Universal Robots URScript: test-1.urscript

def tuft_program():
    global tuft_coords = p[-0.743799, 1.270828, -0.183331, 1.574839, 0.004352, -0.002073]
    global current_pose = p[0,0,0,-1.19353,1.19941,1.24224]
    textmsg("Starting tufting job test-1.jpg")
    textmsg("Using coordinate frame tuft_coords")
    set_digital_out(0, False)
    global travel_speed = 0.2000
    global tuft_speed = 0.0600
    global contact_force_threshold = 15.00
    global contact_probe_step = 0.0010
    global progress_host = "127.0.0.1"
    global progress_port = 4700
    global progress_total = 2256
    global progress_current = 0
    global progress_job_id = "645c90bf-1acd-4e3e-9f73-d32fedb47cbd"
    global open=socket_open(progress_host,progress_port)
    while (open ==  False  ):
        global open=socket_open(progress_host,progress_port)
    end
    def report_progress():
        progress_current = progress_current + 1
        global sendToServer="{jobId:" + progress_job_id + ",current:" + to_str(progress_current) + ",total:" + to_str(progress_total) + "}
"
        socket_send_string(sendToServer)
    end
    new_pose = pose_trans(tuft_coords, p[0.3854, 0.5062, 0.1500, 0, 0, 0])
    movel(p[new_pose[0], new_pose[1], new_pose[2], current_pose[3], current_pose[4], current_pose[5]], a=1.2, v=0.2000)
    report_progress()
    new_pose = pose_trans(tuft_coords, p[0.3854, 0.5062, -0.0020, 0, 0, 0])
    movel(p[new_pose[0], new_pose[1], new_pose[2], current_pose[3], current_pose[4], current_pose[5]], a=0.8, v=0.2000)
    report_progress()
    set_digital_out(0, True)
    new_pose = pose_trans(tuft_coords, p[0.3854, 0.5438, -0.0020, 0, 0, 0])
    movel(p[new_pose[0], new_pose[1], new_pose[2], current_pose[3], current_pose[4], current_pose[5]], a=1.2, v=0.0600)
    report_progress()
    set_digital_out(0, False)
    new_pose = pose_trans(tuft_coords, p[0.3854, 0.5438, 0.1500, 0, 0, 0])
    movel(p[new_pose[0], new_pose[1], new_pose[2], current_pose[3], current_pose[4], current_pose[5]], a=0.8, v=0.2000)
    report_progress()
    new_pose = pose_trans(tuft_coords, p[0.3874, 0.4824, 0.1500, 0, 0, 0])
    movel(p[new_pose[0], new_pose[1], new_pose[2], current_pose[3], current_pose[4], current_pose[5]], a=1.2, v=0.2000)
    report_progress()
    new_pose = pose_trans(tuft_coords, p[0.3874, 0.4824, -0.0020, 0, 0, 0])
    movel(p[new_pose[0], new_pose[1], new_pose[2], current_pose[3], current_pose[4], current_pose[5]], a=0.8, v=0.2000)
    report_progress()
    set_digital_out(0, True)
    new_pose = pose_trans(tuft_coords, p[0.3874, 0.5676, -0.0020, 0, 0, 0])
    movel(p[new_pose[0], new_pose[1], new_pose[2], current_pose[3], current_pose[4], current_pose[5]], a=1.2, v=0.0600)
    report_progress()
    set_digital_out(0, False)
    new_pose = pose_trans(tuft_coords, p[0.3874, 0.5676, 0.1500, 0, 0, 0])
    movel(p[new_pose[0], new_pose[1], new_pose[2], current_pose[3], current_pose[4], current_pose[5]], a=0.8, v=0.2000)
    report_progress()
    new_pose = pose_trans(tuft_coords, p[0.3893, 0.4686, 0.1500, 0, 0, 0])
    movel(p[new_pose[0], new_pose[1], new_pose[2], current_pose[3], current_pose[4], current_pose[5]], a=1.2, v=0.2000)
    report_progress()
    new_pose = pose_trans(tuft_coords, p[0.3893, 0.4686, -0.0020, 0, 0, 0])
    movel(p[new_pose[0], new_pose[1], new_pose[2], current_pose[3], current_pose[4], current_pose[5]], a=0.8, v=0.2000)
    report_progress()
    set_digital_out(0, True)
    new_pose = pose_trans(tuft_coords, p[0.3893, 0.5814, -0.0020, 0, 0, 0])
    movel(p[new_pose[0], new_pose[1], new_pose[2], current_pose[3], current_pose[4], current_pose[5]], a=1.2, v=0.0600)
    report_progress()
    set_digital_out(0, False)
    new_pose = pose_trans(tuft_coords, p[0.3893, 0.5814, 0.1500, 0, 0, 0])
    movel(p[new_pose[0], new_pose[1], new_pose[2], current_pose[3], current_pose[4], current_pose[5]], a=0.8, v=0.2000)
    report_progress()
    new_pose = pose_trans(tuft_coords, p[0.3912, 0.4567, 0.1500, 0, 0, 0])
    movel(p[new_pose[0], new_pose[1], new_pose[2], current_pose[3], current_pose[4], current_pose[5]], a=1.2, v=0.2000)
    report_progress()
    new_pose = pose_trans(tuft_coords, p[0.3912, 0.4567, -0.0020, 0, 0, 0])
    movel(p[new_pose[0], new_pose[1], new_pose[2], current_pose[3], current_pose[4], current_pose[5]], a=0.8, v=0.2000)
    report_progress()
    set_digital_out(0, True)
    new_pose = pose_trans(tuft_coords, p[0.3912, 0.5933, -0.0020, 0, 0, 0])
    movel(p[new_pose[0], new_pose[1], new_pose[2], current_pose[3], current_pose[4], current_pose[5]], a=1.2, v=0.0600)
    report_progress()
    set_digital_out(0, False)
    new_pose = pose_trans(tuft_coords, p[0.3912, 0.5933, 0.1500, 0, 0, 0])
    movel(p[new_pose[0], new_pose[1], new_pose[2], current_pose[3], current_pose[4], current_pose[5]], a=0.8, v=0.2000)
    report_progress()
    new_pose = pose_trans(tuft_coords, p[0.3932, 0.4468, 0.1500, 0, 0, 0])
    movel(p[new_pose[0], new_pose[1], new_pose[2], current_pose[3], current_pose[4], current_pose[5]], a=1.2, v=0.2000)
    report_progress()
    new_pose = pose_trans(tuft_coords, p[0.3932, 0.4468, -0.0020, 0, 0, 0])
    movel(p[new_pose[0], new_pose[1], new_pose[2], current_pose[3], current_pose[4], current_pose[5]], a=0.8, v=0.2000)
    report_progress()
    set_digital_out(0, True)
    new_pose = pose_trans(tuft_coords, p[0.3932, 0.6032, -0.0020, 0, 0, 0])
    movel(p[new_pose[0], new_pose[1], new_pose[2], current_pose[3], current_pose[4], current_pose[5]], a=1.2, v=0.0600)
    report_progress()
    set_digital_out(0, False)
    new_pose = pose_trans(tuft_coords, p[0.3932, 0.6032, 0.1500, 0, 0, 0])
    movel(p[new_pose[0], new_pose[1], new_pose[2], current_pose[3], current_pose[4], current_pose[5]], a=0.8, v=0.2000)
    report_progress()
    new_pose = pose_trans(tuft_coords, p[0.3951, 0.4389, 0.1500, 0, 0, 0])
    movel(p[new_pose[0], new_pose[1], new_pose[2], current_pose[3], current_pose[4], current_pose[5]], a=1.2, v=0.2000)
    report_progress()
    new_pose = pose_trans(tuft_coords, p[0.3951, 0.4389, -0.0020, 0, 0, 0])
    movel(p[new_pose[0], new_pose[1], new_pose[2], current_pose[3], current_pose[4], current_pose[5]], a=0.8, v=0.2000)
    report_progress()
    set_digital_out(0, True)
    new_pose = pose_trans(tuft_coords, p[0.3951, 0.6111, -0.0020, 0, 0, 0])
    movel(p[new_pose[0], new_pose[1], new_pose[2], current_pose[3], current_pose[4], current_pose[5]], a=1.2, v=0.0600)
    report_progress()
    set_digital_out(0, False)
    new_pose = pose_trans(tuft_coords, p[0.3951, 0.6111, 0.1500, 0, 0, 0])
    movel(p[new_pose[0], new_pose[1], new_pose[2], current_pose[3], current_pose[4], current_pose[5]], a=0.8, v=0.2000)
    report_progress()
    new_pose = pose_trans(tuft_coords, p[0.3971, 0.4310, 0.1500, 0, 0, 0])
    movel(p[new_pose[0], new_pose[1], new_pose[2], current_pose[3], current_pose[4], current_pose[5]], a=1.2, v=0.2000)
    report_progress()
    new_pose = pose_trans(tuft_coords, p[0.3971, 0.4310, -0.0020, 0, 0, 0])
    movel(p[new_pose[0], new_pose[1], new_pose[2], current_pose[3], current_pose[4], current_pose[5]], a=0.8, v=0.2000)
    report_progress()
    set_digital_out(0, True)
    new_pose = pose_trans(tuft_coords, p[0.3971, 0.6190, -0.0020, 0, 0, 0])
    movel(p[new_pose[0], new_pose[1], new_pose[2], current_pose[3], current_pose[4], current_pose[5]], a=1.2, v=0.0600)
    report_progress()
    set_digital_out(0, False)
    new_pose = pose_trans(tuft_coords, p[0.3971, 0.6190, 0.1500, 0, 0, 0])
    movel(p[new_pose[0], new_pose[1], new_pose[2], current_pose[3], current_pose[4], current_pose[5]], a=0.8, v=0.2000)
    report_progress()
    new_pose = pose_trans(tuft_coords, p[0.3990, 0.4231, 0.1500, 0, 0, 0])
    movel(p[new_pose[0], new_pose[1], new_pose[2], current_pose[3], current_pose[4], current_pose[5]], a=1.2, v=0.2000)
    report_progress()
    new_pose = pose_trans(tuft_coords, p[0.3990, 0.4231, -0.0020, 0, 0, 0])
    movel(p[new_pose[0], new_pose[1], new_pose[2], current_pose[3], current_pose[4], current_pose[5]], a=0.8, v=0.2000)
    report_progress()
    set_digital_out(0, True)
    new_pose = pose_trans(tuft_coords, p[0.3990, 0.6269, -0.0020, 0, 0, 0])
    movel(p[new_pose[0], new_pose[1], new_pose[2], current_pose[3], current_pose[4], current_pose[5]], a=1.2, v=0.0600)
    report_progress()
    set_digital_out(0, False)
    new_pose = pose_trans(tuft_coords, p[0.3990, 0.6269, 0.1500, 0, 0, 0])
    movel(p[new_pose[0], new_pose[1], new_pose[2], current_pose[3], current_pose[4], current_pose[5]], a=0.8, v=0.2000)
    report_progress()
    new_pose = pose_trans(tuft_coords, p[0.4010, 0.4171, 0.1500, 0, 0, 0])
    movel(p[new_pose[0], new_pose[1], new_pose[2], current_pose[3], current_pose[4], current_pose[5]], a=1.2, v=0.2000)
    report_progress()
    new_pose = pose_trans(tuft_coords, p[0.4010, 0.4171, -0.0020, 0, 0, 0])
    movel(p[new_pose[0], new_pose[1], new_pose[2], current_pose[3], current_pose[4], current_pose[5]], a=0.8, v=0.2000)
    report_progress()
    set_digital_out(0, True)
    new_pose = pose_trans(tuft_coords, p[0.4010, 0.6329, -0.0020, 0, 0, 0])
    movel(p[new_pose[0], new_pose[1], new_pose[2], current_pose[3], current_pose[4], current_pose[5]], a=1.2, v=0.0600)
    report_progress()
    set_digital_out(0, False)
    new_pose = pose_trans(tuft_coords, p[0.4010, 0.6329, 0.1500, 0, 0, 0])
    movel(p[new_pose[0], new_pose[1], new_pose[2], current_pose[3], current_pose[4], current_pose[5]], a=0.8, v=0.2000)
    report_progress()
    new_pose = pose_trans(tuft_coords, p[0.4029, 0.4112, 0.1500, 0, 0, 0])
    movel(p[new_pose[0], new_pose[1], new_pose[2], current_pose[3], current_pose[4], current_pose[5]], a=1.2, v=0.2000)
    report_progress()
    new_pose = pose_trans(tuft_coords, p[0.4029, 0.4112, -0.0020, 0, 0, 0])
    movel(p[new_pose[0], new_pose[1], new_pose[2], current_pose[3], current_pose[4], current_pose[5]], a=0.8, v=0.2000)
    report_progress()
    set_digital_out(0, True)
    new_pose = pose_trans(tuft_coords, p[0.4029, 0.6388, -0.0020, 0, 0, 0])
    movel(p[new_pose[0], new_pose[1], new_pose[2], current_pose[3], current_pose[4], current_pose[5]], a=1.2, v=0.0600)
    report_progress()
    set_digital_out(0, False)
    new_pose = pose_trans(tuft_coords, p[0.4029, 0.6388, 0.1500, 0, 0, 0])
    movel(p[new_pose[0], new_pose[1], new_pose[2], current_pose[3], current_pose[4], current_pose[5]], a=0.8, v=0.2000)
    report_progress()
    new_pose = pose_trans(tuft_coords, p[0.4049, 0.4053, 0.1500, 0, 0, 0])
    movel(p[new_pose[0], new_pose[1], new_pose[2], current_pose[3], current_pose[4], current_pose[5]], a=1.2, v=0.2000)
    report_progress()
    new_pose = pose_trans(tuft_coords, p[0.4049, 0.4053, -0.0020, 0, 0, 0])
    movel(p[new_pose[0], new_pose[1], new_pose[2], current_pose[3], current_pose[4], current_pose[5]], a=0.8, v=0.2000)
    report_progress()
    set_digital_out(0, True)
    new_pose = pose_trans(tuft_coords, p[0.4049, 0.6447, -0.0020, 0, 0, 0])
    movel(p[new_pose[0], new_pose[1], new_pose[2], current_pose[3], current_pose[4], current_pose[5]], a=1.2, v=0.0600)
    report_progress()
    set_digital_out(0, False)
    new_pose = pose_trans(tuft_coords, p[0.4049, 0.6447, 0.1500, 0, 0, 0])
    movel(p[new_pose[0], new_pose[1], new_pose[2], current_pose[3], current_pose[4], current_pose[5]], a=0.8, v=0.2000)
    report_progress()
    new_pose = pose_trans(tuft_coords, p[0.4068, 0.3993, 0.1500, 0, 0, 0])
    movel(p[new_pose[0], new_pose[1], new_pose[2], current_pose[3], current_pose[4], current_pose[5]], a=1.2, v=0.2000)
    report_progress()
    new_pose = pose_trans(tuft_coords, p[0.4068, 0.3993, -0.0020, 0, 0, 0])
    movel(p[new_pose[0], new_pose[1], new_pose[2], current_pose[3], current_pose[4], current_pose[5]], a=0.8, v=0.2000)
    report_progress()
    set_digital_out(0, True)
    new_pose = pose_trans(tuft_coords, p[0.4068, 0.6507, -0.0020, 0, 0, 0])
    movel(p[new_pose[0], new_pose[1], new_pose[2], current_pose[3], current_pose[4], current_pose[5]], a=1.2, v=0.0600)
    report_progress()
    set_digital_out(0, False)
    new_pose = pose_trans(tuft_coords, p[0.4068, 0.6507, 0.1500, 0, 0, 0])
    movel(p[new_pose[0], new_pose[1], new_pose[2], current_pose[3], current_pose[4], current_pose[5]], a=0.8, v=0.2000)
    report_progress()
    new_pose = pose_trans(tuft_coords, p[0.4088, 0.3934, 0.1500, 0, 0, 0])
    movel(p[new_pose[0], new_pose[1], new_pose[2], current_pose[3], current_pose[4], current_pose[5]], a=1.2, v=0.2000)
    report_progress()
    new_pose = pose_trans(tuft_coords, p[0.4088, 0.3934, -0.0020, 0, 0, 0])
    movel(p[new_pose[0], new_pose[1], new_pose[2], current_pose[3], current_pose[4], current_pose[5]], a=0.8, v=0.2000)
    report_progress()
    set_digital_out(0, True)
    new_pose = pose_trans(tuft_coords, p[0.4088, 0.6566, -0.0020, 0, 0, 0])
    movel(p[new_pose[0], new_pose[1], new_pose[2], current_pose[3], current_pose[4], current_pose[5]], a=1.2, v=0.0600)
    report_progress()
    set_digital_out(0, False)
    new_pose = pose_trans(tuft_coords, p[0.4088, 0.6566, 0.1500, 0, 0, 0])
    movel(p[new_pose[0], new_pose[1], new_pose[2], current_pose[3], current_pose[4], current_pose[5]], a=0.8, v=0.2000)
    report_progress()
    new_pose = pose_trans(tuft_coords, p[0.4107, 0.3874, 0.1500, 0, 0, 0])
    movel(p[new_pose[0], new_pose[1], new_pose[2], current_pose[3], current_pose[4], current_pose[5]], a=1.2, v=0.2000)
    report_progress()
    new_pose = pose_trans(tuft_coords, p[0.4107, 0.3874, -0.0020, 0, 0, 0])
    movel(p[new_pose[0], new_pose[1], new_pose[2], current_pose[3], current_pose[4], current_pose[5]], a=0.8, v=0.2000)
    report_progress()
    set_digital_out(0, True)
    new_pose = pose_trans(tuft_coords, p[0.4107, 0.6606, -0.0020, 0, 0, 0])
    movel(p[new_pose[0], new_pose[1], new_pose[2], current_pose[3], current_pose[4], current_pose[5]], a=1.2, v=0.0600)
    report_progress()
    set_digital_out(0, False)
    new_pose = pose_trans(tuft_coords, p[0.4107, 0.6606, 0.1500, 0, 0, 0])
    movel(p[new_pose[0], new_pose[1], new_pose[2], current_pose[3], current_pose[4], current_pose[5]], a=0.8, v=0.2000)
    report_progress()
    new_pose = pose_trans(tuft_coords, p[0.4126, 0.3835, 0.1500, 0, 0, 0])
    movel(p[new_pose[0], new_pose[1], new_pose[2], current_pose[3], current_pose[4], current_pose[5]], a=1.2, v=0.2000)
    report_progress()
    new_pose = pose_trans(tuft_coords, p[0.4126, 0.3835, -0.0020, 0, 0, 0])
    movel(p[new_pose[0], new_pose[1], new_pose[2], current_pose[3], current_pose[4], current_pose[5]], a=0.8, v=0.2000)
    report_progress()
    set_digital_out(0, True)
    new_pose = pose_trans(tuft_coords, p[0.4126, 0.6665, -0.0020, 0, 0, 0])
    movel(p[new_pose[0], new_pose[1], new_pose[2], current_pose[3], current_pose[4], current_pose[5]], a=1.2, v=0.0600)
    report_progress()
    set_digital_out(0, False)
    new_pose = pose_trans(tuft_coords, p[0.4126, 0.6665, 0.1500, 0, 0, 0])
    movel(p[new_pose[0], new_pose[1], new_pose[2], current_pose[3], current_pose[4], current_pose[5]], a=0.8, v=0.2000)
    report_progress()
    new_pose = pose_trans(tuft_coords, p[0.4146, 0.3795, 0.1500, 0, 0, 0])
    movel(p[new_pose[0], new_pose[1], new_pose[2], current_pose[3], current_pose[4], current_pose[5]], a=1.2, v=0.2000)
    report_progress()
    new_pose = pose_trans(tuft_coords, p[0.4146, 0.3795, -0.0020, 0, 0, 0])
    movel(p[new_pose[0], new_pose[1], new_pose[2], current_pose[3], current_pose[4], current_pose[5]], a=0.8, v=0.2000)
    report_progress()
    set_digital_out(0, True)
    new_pose = pose_trans(tuft_coords, p[0.4146, 0.6705, -0.0020, 0, 0, 0])
    movel(p[new_pose[0], new_pose[1], new_pose[2], current_pose[3], current_pose[4], current_pose[5]], a=1.2, v=0.0600)
    report_progress()
    set_digital_out(0, False)
    new_pose = pose_trans(tuft_coords, p[0.4146, 0.6705, 0.1500, 0, 0, 0])
    movel(p[new_pose[0], new_pose[1], new_pose[2], current_pose[3], current_pose[4], current_pose[5]], a=0.8, v=0.2000)
    report_progress()
    new_pose = pose_trans(tuft_coords, p[0.4165, 0.3736, 0.1500, 0, 0, 0])
    movel(p[new_pose[0], new_pose[1], new_pose[2], current_pose[3], current_pose[4], current_pose[5]], a=1.2, v=0.2000)
    report_progress()
    new_pose = pose_trans(tuft_coords, p[0.4165, 0.3736, -0.0020, 0, 0, 0])
    movel(p[new_pose[0], new_pose[1], new_pose[2], current_pose[3], current_pose[4], current_pose[5]], a=0.8, v=0.2000)
    report_progress()
    set_digital_out(0, True)
    new_pose = pose_trans(tuft_coords, p[0.4165, 0.6764, -0.0020, 0, 0, 0])
    movel(p[new_pose[0], new_pose[1], new_pose[2], current_pose[3], current_pose[4], current_pose[5]], a=1.2, v=0.0600)
    report_progress()
    set_digital_out(0, False)
    new_pose = pose_trans(tuft_coords, p[0.4165, 0.6764, 0.1500, 0, 0, 0])
    movel(p[new_pose[0], new_pose[1], new_pose[2], current_pose[3], current_pose[4], current_pose[5]], a=0.8, v=0.2000)
    report_progress()
    new_pose = pose_trans(tuft_coords, p[0.4185, 0.3696, 0.1500, 0, 0, 0])
    movel(p[new_pose[0], new_pose[1], new_pose[2], current_pose[3], current_pose[4], current_pose[5]], a=1.2, v=0.2000)
    report_progress()
    new_pose = pose_trans(tuft_coords, p[0.4185, 0.3696, -0.0020, 0, 0, 0])
    movel(p[new_pose[0], new_pose[1], new_pose[2], current_pose[3], current_pose[4], current_pose[5]], a=0.8, v=0.2000)
    report_progress()
    set_digital_out(0, True)
    new_pose = pose_trans(tuft_coords, p[0.4185, 0.6804, -0.0020, 0, 0, 0])
    movel(p[new_pose[0], new_pose[1], new_pose[2], current_pose[3], current_pose[4], current_pose[5]], a=1.2, v=0.0600)
    report_progress()
    set_digital_out(0, False)
    new_pose = pose_trans(tuft_coords, p[0.4185, 0.6804, 0.1500, 0, 0, 0])
    movel(p[new_pose[0], new_pose[1], new_pose[2], current_pose[3], current_pose[4], current_pose[5]], a=0.8, v=0.2000)
    report_progress()
    new_pose = pose_trans(tuft_coords, p[0.4204, 0.3657, 0.1500, 0, 0, 0])
    movel(p[new_pose[0], new_pose[1], new_pose[2], current_pose[3], current_pose[4], current_pose[5]], a=1.2, v=0.2000)
    report_progress()
    new_pose = pose_trans(tuft_coords, p[0.4204, 0.3657, -0.0020, 0, 0, 0])
    movel(p[new_pose[0], new_pose[1], new_pose[2], current_pose[3], current_pose[4], current_pose[5]], a=0.8, v=0.2000)
    report_progress()
    set_digital_out(0, True)
    new_pose = pose_trans(tuft_coords, p[0.4204, 0.6843, -0.0020, 0, 0, 0])
    movel(p[new_pose[0], new_pose[1], new_pose[2], current_pose[3], current_pose[4], current_pose[5]], a=1.2, v=0.0600)
    report_progress()
    set_digital_out(0, False)
    new_pose = pose_trans(tuft_coords, p[0.4204, 0.6843, 0.1500, 0, 0, 0])
    movel(p[new_pose[0], new_pose[1], new_pose[2], current_pose[3], current_pose[4], current_pose[5]], a=0.8, v=0.2000)
    report_progress()
    new_pose = pose_trans(tuft_coords, p[0.4224, 0.3617, 0.1500, 0, 0, 0])
    movel(p[new_pose[0], new_pose[1], new_pose[2], current_pose[3], current_pose[4], current_pose[5]], a=1.2, v=0.2000)
    report_progress()
    new_pose = pose_trans(tuft_coords, p[0.4224, 0.3617, -0.0020, 0, 0, 0])
    movel(p[new_pose[0], new_pose[1], new_pose[2], current_pose[3], current_pose[4], current_pose[5]], a=0.8, v=0.2000)
    report_progress()
    set_digital_out(0, True)
    new_pose = pose_trans(tuft_coords, p[0.4224, 0.6883, -0.0020, 0, 0, 0])
    movel(p[new_pose[0], new_pose[1], new_pose[2], current_pose[3], current_pose[4], current_pose[5]], a=1.2, v=0.0600)
    report_progress()
    set_digital_out(0, False)
    new_pose = pose_trans(tuft_coords, p[0.4224, 0.6883, 0.1500, 0, 0, 0])
    movel(p[new_pose[0], new_pose[1], new_pose[2], current_pose[3], current_pose[4], current_pose[5]], a=0.8, v=0.2000)
    report_progress()
    new_pose = pose_trans(tuft_coords, p[0.4243, 0.3578, 0.1500, 0, 0, 0])
    movel(p[new_pose[0], new_pose[1], new_pose[2], current_pose[3], current_pose[4], current_pose[5]], a=1.2, v=0.2000)
    report_progress()
    new_pose = pose_trans(tuft_coords, p[0.4243, 0.3578, -0.0020, 0, 0, 0])
    movel(p[new_pose[0], new_pose[1], new_pose[2], current_pose[3], current_pose[4], current_pose[5]], a=0.8, v=0.2000)
    report_progress()
    set_digital_out(0, True)
    new_pose = pose_trans(tuft_coords, p[0.4243, 0.6922, -0.0020, 0, 0, 0])
    movel(p[new_pose[0], new_pose[1], new_pose[2], current_pose[3], current_pose[4], current_pose[5]], a=1.2, v=0.0600)
    report_progress()
    set_digital_out(0, False)
    new_pose = pose_trans(tuft_coords, p[0.4243, 0.6922, 0.1500, 0, 0, 0])
    movel(p[new_pose[0], new_pose[1], new_pose[2], current_pose[3], current_pose[4], current_pose[5]], a=0.8, v=0.2000)
    report_progress()
    new_pose = pose_trans(tuft_coords, p[0.4263, 0.3538, 0.1500, 0, 0, 0])
    movel(p[new_pose[0], new_pose[1], new_pose[2], current_pose[3], current_pose[4], current_pose[5]], a=1.2, v=0.2000)
    report_progress()
    new_pose = pose_trans(tuft_coords, p[0.4263, 0.3538, -0.0020, 0, 0, 0])
    movel(p[new_pose[0], new_pose[1], new_pose[2], current_pose[3], current_pose[4], current_pose[5]], a=0.8, v=0.2000)
    report_progress()
    set_digital_out(0, True)
    new_pose = pose_trans(tuft_coords, p[0.4263, 0.6962, -0.0020, 0, 0, 0])
    movel(p[new_pose[0], new_pose[1], new_pose[2], current_pose[3], current_pose[4], current_pose[5]], a=1.2, v=0.0600)
    report_progress()
    set_digital_out(0, False)
    new_pose = pose_trans(tuft_coords, p[0.4263, 0.6962, 0.1500, 0, 0, 0])
    movel(p[new_pose[0], new_pose[1], new_pose[2], current_pose[3], current_pose[4], current_pose[5]], a=0.8, v=0.2000)
    report_progress()
    new_pose = pose_trans(tuft_coords, p[0.4282, 0.3498, 0.1500, 0, 0, 0])
    movel(p[new_pose[0], new_pose[1], new_pose[2], current_pose[3], current_pose[4], current_pose[5]], a=1.2, v=0.2000)
    report_progress()
    new_pose = pose_trans(tuft_coords, p[0.4282, 0.3498, -0.0020, 0, 0, 0])
    movel(p[new_pose[0], new_pose[1], new_pose[2], current_pose[3], current_pose[4], current_pose[5]], a=0.8, v=0.2000)
    report_progress()
    set_digital_out(0, True)
    new_pose = pose_trans(tuft_coords, p[0.4282, 0.7002, -0.0020, 0, 0, 0])
    movel(p[new_pose[0], new_pose[1], new_pose[2], current_pose[3], current_pose[4], current_pose[5]], a=1.2, v=0.0600)
    report_progress()
    set_digital_out(0, False)
    new_pose = pose_trans(tuft_coords, p[0.4282, 0.7002, 0.1500, 0, 0, 0])
    movel(p[new_pose[0], new_pose[1], new_pose[2], current_pose[3], current_pose[4], current_pose[5]], a=0.8, v=0.2000)
    report_progress()
    new_pose = pose_trans(tuft_coords, p[0.4301, 0.3459, 0.1500, 0, 0, 0])
    movel(p[new_pose[0], new_pose[1], new_pose[2], current_pose[3], current_pose[4], current_pose[5]], a=1.2, v=0.2000)
    report_progress()
    new_pose = pose_trans(tuft_coords, p[0.4301, 0.3459, -0.0020, 0, 0, 0])
    movel(p[new_pose[0], new_pose[1], new_pose[2], current_pose[3], current_pose[4], current_pose[5]], a=0.8, v=0.2000)
    report_progress()
    set_digital_out(0, True)
    new_pose = pose_trans(tuft_coords, p[0.4301, 0.7041, -0.0020, 0, 0, 0])
    movel(p[new_pose[0], new_pose[1], new_pose[2], current_pose[3], current_pose[4], current_pose[5]], a=1.2, v=0.0600)
    report_progress()
    set_digital_out(0, False)
    new_pose = pose_trans(tuft_coords, p[0.4301, 0.7041, 0.1500, 0, 0, 0])
    movel(p[new_pose[0], new_pose[1], new_pose[2], current_pose[3], current_pose[4], current_pose[5]], a=0.8, v=0.2000)
    report_progress()
    new_pose = pose_trans(tuft_coords, p[0.4321, 0.3439, 0.1500, 0, 0, 0])
    movel(p[new_pose[0], new_pose[1], new_pose[2], current_pose[3], current_pose[4], current_pose[5]], a=1.2, v=0.2000)
    report_progress()
    new_pose = pose_trans(tuft_coords, p[0.4321, 0.3439, -0.0020, 0, 0, 0])
    movel(p[new_pose[0], new_pose[1], new_pose[2], current_pose[3], current_pose[4], current_pose[5]], a=0.8, v=0.2000)
    report_progress()
    set_digital_out(0, True)
    new_pose = pose_trans(tuft_coords, p[0.4321, 0.7061, -0.0020, 0, 0, 0])
    movel(p[new_pose[0], new_pose[1], new_pose[2], current_pose[3], current_pose[4], current_pose[5]], a=1.2, v=0.0600)
    report_progress()
    set_digital_out(0, False)
    new_pose = pose_trans(tuft_coords, p[0.4321, 0.7061, 0.1500, 0, 0, 0])
    movel(p[new_pose[0], new_pose[1], new_pose[2], current_pose[3], current_pose[4], current_pose[5]], a=0.8, v=0.2000)
    report_progress()
    new_pose = pose_trans(tuft_coords, p[0.4340, 0.3399, 0.1500, 0, 0, 0])
    movel(p[new_pose[0], new_pose[1], new_pose[2], current_pose[3], current_pose[4], current_pose[5]], a=1.2, v=0.2000)
    report_progress()
    new_pose = pose_trans(tuft_coords, p[0.4340, 0.3399, -0.0020, 0, 0, 0])
    movel(p[new_pose[0], new_pose[1], new_pose[2], current_pose[3], current_pose[4], current_pose[5]], a=0.8, v=0.2000)
    report_progress()
    set_digital_out(0, True)
    new_pose = pose_trans(tuft_coords, p[0.4340, 0.7101, -0.0020, 0, 0, 0])
    movel(p[new_pose[0], new_pose[1], new_pose[2], current_pose[3], current_pose[4], current_pose[5]], a=1.2, v=0.0600)
    report_progress()
    set_digital_out(0, False)
    new_pose = pose_trans(tuft_coords, p[0.4340, 0.7101, 0.1500, 0, 0, 0])
    movel(p[new_pose[0], new_pose[1], new_pose[2], current_pose[3], current_pose[4], current_pose[5]], a=0.8, v=0.2000)
    report_progress()
    new_pose = pose_trans(tuft_coords, p[0.4360, 0.3360, 0.1500, 0, 0, 0])
    movel(p[new_pose[0], new_pose[1], new_pose[2], current_pose[3], current_pose[4], current_pose[5]], a=1.2, v=0.2000)
    report_progress()
    new_pose = pose_trans(tuft_coords, p[0.4360, 0.3360, -0.0020, 0, 0, 0])
    movel(p[new_pose[0], new_pose[1], new_pose[2], current_pose[3], current_pose[4], current_pose[5]], a=0.8, v=0.2000)
    report_progress()
    set_digital_out(0, True)
    new_pose = pose_trans(tuft_coords, p[0.4360, 0.7140, -0.0020, 0, 0, 0])
    movel(p[new_pose[0], new_pose[1], new_pose[2], current_pose[3], current_pose[4], current_pose[5]], a=1.2, v=0.0600)
    report_progress()
    set_digital_out(0, False)
    new_pose = pose_trans(tuft_coords, p[0.4360, 0.7140, 0.1500, 0, 0, 0])
    movel(p[new_pose[0], new_pose[1], new_pose[2], current_pose[3], current_pose[4], current_pose[5]], a=0.8, v=0.2000)
    report_progress()
    new_pose = pose_trans(tuft_coords, p[0.4379, 0.3340, 0.1500, 0, 0, 0])
    movel(p[new_pose[0], new_pose[1], new_pose[2], current_pose[3], current_pose[4], current_pose[5]], a=1.2, v=0.2000)
    report_progress()
    new_pose = pose_trans(tuft_coords, p[0.4379, 0.3340, -0.0020, 0, 0, 0])
    movel(p[new_pose[0], new_pose[1], new_pose[2], current_pose[3], current_pose[4], current_pose[5]], a=0.8, v=0.2000)
    report_progress()
    set_digital_out(0, True)
    new_pose = pose_trans(tuft_coords, p[0.4379, 0.7160, -0.0020, 0, 0, 0])
    movel(p[new_pose[0], new_pose[1], new_pose[2], current_pose[3], current_pose[4], current_pose[5]], a=1.2, v=0.0600)
    report_progress()
    set_digital_out(0, False)
    new_pose = pose_trans(tuft_coords, p[0.4379, 0.7160, 0.1500, 0, 0, 0])
    movel(p[new_pose[0], new_pose[1], new_pose[2], current_pose[3], current_pose[4], current_pose[5]], a=0.8, v=0.2000)
    report_progress()
    new_pose = pose_trans(tuft_coords, p[0.4399, 0.3301, 0.1500, 0, 0, 0])
    movel(p[new_pose[0], new_pose[1], new_pose[2], current_pose[3], current_pose[4], current_pose[5]], a=1.2, v=0.2000)
    report_progress()
    new_pose = pose_trans(tuft_coords, p[0.4399, 0.3301, -0.0020, 0, 0, 0])
    movel(p[new_pose[0], new_pose[1], new_pose[2], current_pose[3], current_pose[4], current_pose[5]], a=0.8, v=0.2000)
    report_progress()
    set_digital_out(0, True)
    new_pose = pose_trans(tuft_coords, p[0.4399, 0.7199, -0.0020, 0, 0, 0])
    movel(p[new_pose[0], new_pose[1], new_pose[2], current_pose[3], current_pose[4], current_pose[5]], a=1.2, v=0.0600)
    report_progress()
    set_digital_out(0, False)
    new_pose = pose_trans(tuft_coords, p[0.4399, 0.7199, 0.1500, 0, 0, 0])
    movel(p[new_pose[0], new_pose[1], new_pose[2], current_pose[3], current_pose[4], current_pose[5]], a=0.8, v=0.2000)
    report_progress()
    new_pose = pose_trans(tuft_coords, p[0.4418, 0.3261, 0.1500, 0, 0, 0])
    movel(p[new_pose[0], new_pose[1], new_pose[2], current_pose[3], current_pose[4], current_pose[5]], a=1.2, v=0.2000)
    report_progress()
    new_pose = pose_trans(tuft_coords, p[0.4418, 0.3261, -0.0020, 0, 0, 0])
    movel(p[new_pose[0], new_pose[1], new_pose[2], current_pose[3], current_pose[4], current_pose[5]], a=0.8, v=0.2000)
    report_progress()
    set_digital_out(0, True)
    new_pose = pose_trans(tuft_coords, p[0.4418, 0.7239, -0.0020, 0, 0, 0])
    movel(p[new_pose[0], new_pose[1], new_pose[2], current_pose[3], current_pose[4], current_pose[5]], a=1.2, v=0.0600)
    report_progress()
    set_digital_out(0, False)
    new_pose = pose_trans(tuft_coords, p[0.4418, 0.7239, 0.1500, 0, 0, 0])
    movel(p[new_pose[0], new_pose[1], new_pose[2], current_pose[3], current_pose[4], current_pose[5]], a=0.8, v=0.2000)
    report_progress()
    new_pose = pose_trans(tuft_coords, p[0.4437, 0.3241, 0.1500, 0, 0, 0])
    movel(p[new_pose[0], new_pose[1], new_pose[2], current_pose[3], current_pose[4], current_pose[5]], a=1.2, v=0.2000)
    report_progress()
    new_pose = pose_trans(tuft_coords, p[0.4437, 0.3241, -0.0020, 0, 0, 0])
    movel(p[new_pose[0], new_pose[1], new_pose[2], current_pose[3], current_pose[4], current_pose[5]], a=0.8, v=0.2000)
    report_progress()
    set_digital_out(0, True)
    new_pose = pose_trans(tuft_coords, p[0.4437, 0.7259, -0.0020, 0, 0, 0])
    movel(p[new_pose[0], new_pose[1], new_pose[2], current_pose[3], current_pose[4], current_pose[5]], a=1.2, v=0.0600)
    report_progress()
    set_digital_out(0, False)
    new_pose = pose_trans(tuft_coords, p[0.4437, 0.7259, 0.1500, 0, 0, 0])
    movel(p[new_pose[0], new_pose[1], new_pose[2], current_pose[3], current_pose[4], current_pose[5]], a=0.8, v=0.2000)
    report_progress()
    new_pose = pose_trans(tuft_coords, p[0.4457, 0.3202, 0.1500, 0, 0, 0])
    movel(p[new_pose[0], new_pose[1], new_pose[2], current_pose[3], current_pose[4], current_pose[5]], a=1.2, v=0.2000)
    report_progress()
    new_pose = pose_trans(tuft_coords, p[0.4457, 0.3202, -0.0020, 0, 0, 0])
    movel(p[new_pose[0], new_pose[1], new_pose[2], current_pose[3], current_pose[4], current_pose[5]], a=0.8, v=0.2000)
    report_progress()
    set_digital_out(0, True)
    new_pose = pose_trans(tuft_coords, p[0.4457, 0.7298, -0.0020, 0, 0, 0])
    movel(p[new_pose[0], new_pose[1], new_pose[2], current_pose[3], current_pose[4], current_pose[5]], a=1.2, v=0.0600)
    report_progress()
    set_digital_out(0, False)
    new_pose = pose_trans(tuft_coords, p[0.4457, 0.7298, 0.1500, 0, 0, 0])
    movel(p[new_pose[0], new_pose[1], new_pose[2], current_pose[3], current_pose[4], current_pose[5]], a=0.8, v=0.2000)
    report_progress()
    new_pose = pose_trans(tuft_coords, p[0.4476, 0.3182, 0.1500, 0, 0, 0])
    movel(p[new_pose[0], new_pose[1], new_pose[2], current_pose[3], current_pose[4], current_pose[5]], a=1.2, v=0.2000)
    report_progress()
    new_pose = pose_trans(tuft_coords, p[0.4476, 0.3182, -0.0020, 0, 0, 0])
    movel(p[new_pose[0], new_pose[1], new_pose[2], current_pose[3], current_pose[4], current_pose[5]], a=0.8, v=0.2000)
    report_progress()
    set_digital_out(0, True)
    new_pose = pose_trans(tuft_coords, p[0.4476, 0.7318, -0.0020, 0, 0, 0])
    movel(p[new_pose[0], new_pose[1], new_pose[2], current_pose[3], current_pose[4], current_pose[5]], a=1.2, v=0.0600)
    report_progress()
    set_digital_out(0, False)
    new_pose = pose_trans(tuft_coords, p[0.4476, 0.7318, 0.1500, 0, 0, 0])
    movel(p[new_pose[0], new_pose[1], new_pose[2], current_pose[3], current_pose[4], current_pose[5]], a=0.8, v=0.2000)
    report_progress()
    new_pose = pose_trans(tuft_coords, p[0.4496, 0.3142, 0.1500, 0, 0, 0])
    movel(p[new_pose[0], new_pose[1], new_pose[2], current_pose[3], current_pose[4], current_pose[5]], a=1.2, v=0.2000)
    report_progress()
    new_pose = pose_trans(tuft_coords, p[0.4496, 0.3142, -0.0020, 0, 0, 0])
    movel(p[new_pose[0], new_pose[1], new_pose[2], current_pose[3], current_pose[4], current_pose[5]], a=0.8, v=0.2000)
    report_progress()
    set_digital_out(0, True)
    new_pose = pose_trans(tuft_coords, p[0.4496, 0.7358, -0.0020, 0, 0, 0])
    movel(p[new_pose[0], new_pose[1], new_pose[2], current_pose[3], current_pose[4], current_pose[5]], a=1.2, v=0.0600)
    report_progress()
    set_digital_out(0, False)
    new_pose = pose_trans(tuft_coords, p[0.4496, 0.7358, 0.1500, 0, 0, 0])
    movel(p[new_pose[0], new_pose[1], new_pose[2], current_pose[3], current_pose[4], current_pose[5]], a=0.8, v=0.2000)
    report_progress()
    new_pose = pose_trans(tuft_coords, p[0.4515, 0.3122, 0.1500, 0, 0, 0])
    movel(p[new_pose[0], new_pose[1], new_pose[2], current_pose[3], current_pose[4], current_pose[5]], a=1.2, v=0.2000)
    report_progress()
    new_pose = pose_trans(tuft_coords, p[0.4515, 0.3122, -0.0020, 0, 0, 0])
    movel(p[new_pose[0], new_pose[1], new_pose[2], current_pose[3], current_pose[4], current_pose[5]], a=0.8, v=0.2000)
    report_progress()
    set_digital_out(0, True)
    new_pose = pose_trans(tuft_coords, p[0.4515, 0.7378, -0.0020, 0, 0, 0])
    movel(p[new_pose[0], new_pose[1], new_pose[2], current_pose[3], current_pose[4], current_pose[5]], a=1.2, v=0.0600)
    report_progress()
    set_digital_out(0, False)
    new_pose = pose_trans(tuft_coords, p[0.4515, 0.7378, 0.1500, 0, 0, 0])
    movel(p[new_pose[0], new_pose[1], new_pose[2], current_pose[3], current_pose[4], current_pose[5]], a=0.8, v=0.2000)
    report_progress()
    new_pose = pose_trans(tuft_coords, p[0.4535, 0.3083, 0.1500, 0, 0, 0])
    movel(p[new_pose[0], new_pose[1], new_pose[2], current_pose[3], current_pose[4], current_pose[5]], a=1.2, v=0.2000)
    report_progress()
    new_pose = pose_trans(tuft_coords, p[0.4535, 0.3083, -0.0020, 0, 0, 0])
    movel(p[new_pose[0], new_pose[1], new_pose[2], current_pose[3], current_pose[4], current_pose[5]], a=0.8, v=0.2000)
    report_progress()
    set_digital_out(0, True)
    new_pose = pose_trans(tuft_coords, p[0.4535, 0.7417, -0.0020, 0, 0, 0])
    movel(p[new_pose[0], new_pose[1], new_pose[2], current_pose[3], current_pose[4], current_pose[5]], a=1.2, v=0.0600)
    report_progress()
    set_digital_out(0, False)
    new_pose = pose_trans(tuft_coords, p[0.4535, 0.7417, 0.1500, 0, 0, 0])
    movel(p[new_pose[0], new_pose[1], new_pose[2], current_pose[3], current_pose[4], current_pose[5]], a=0.8, v=0.2000)
    report_progress()
    new_pose = pose_trans(tuft_coords, p[0.4554, 0.3063, 0.1500, 0, 0, 0])
    movel(p[new_pose[0], new_pose[1], new_pose[2], current_pose[3], current_pose[4], current_pose[5]], a=1.2, v=0.2000)
    report_progress()
    new_pose = pose_trans(tuft_coords, p[0.4554, 0.3063, -0.0020, 0, 0, 0])
    movel(p[new_pose[0], new_pose[1], new_pose[2], current_pose[3], current_pose[4], current_pose[5]], a=0.8, v=0.2000)
    report_progress()
    set_digital_out(0, True)
    new_pose = pose_trans(tuft_coords, p[0.4554, 0.7437, -0.0020, 0, 0, 0])
    movel(p[new_pose[0], new_pose[1], new_pose[2], current_pose[3], current_pose[4], current_pose[5]], a=1.2, v=0.0600)
    report_progress()
    set_digital_out(0, False)
    new_pose = pose_trans(tuft_coords, p[0.4554, 0.7437, 0.1500, 0, 0, 0])
    movel(p[new_pose[0], new_pose[1], new_pose[2], current_pose[3], current_pose[4], current_pose[5]], a=0.8, v=0.2000)
    report_progress()
    new_pose = pose_trans(tuft_coords, p[0.4574, 0.3043, 0.1500, 0, 0, 0])
    movel(p[new_pose[0], new_pose[1], new_pose[2], current_pose[3], current_pose[4], current_pose[5]], a=1.2, v=0.2000)
    report_progress()
    new_pose = pose_trans(tuft_coords, p[0.4574, 0.3043, -0.0020, 0, 0, 0])
    movel(p[new_pose[0], new_pose[1], new_pose[2], current_pose[3], current_pose[4], current_pose[5]], a=0.8, v=0.2000)
    report_progress()
    set_digital_out(0, True)
    new_pose = pose_trans(tuft_coords, p[0.4574, 0.7457, -0.0020, 0, 0, 0])
    movel(p[new_pose[0], new_pose[1], new_pose[2], current_pose[3], current_pose[4], current_pose[5]], a=1.2, v=0.0600)
    report_progress()
    set_digital_out(0, False)
    new_pose = pose_trans(tuft_coords, p[0.4574, 0.7457, 0.1500, 0, 0, 0])
    movel(p[new_pose[0], new_pose[1], new_pose[2], current_pose[3], current_pose[4], current_pose[5]], a=0.8, v=0.2000)
    report_progress()
    new_pose = pose_trans(tuft_coords, p[0.4593, 0.3004, 0.1500, 0, 0, 0])
    movel(p[new_pose[0], new_pose[1], new_pose[2], current_pose[3], current_pose[4], current_pose[5]], a=1.2, v=0.2000)
    report_progress()
    new_pose = pose_trans(tuft_coords, p[0.4593, 0.3004, -0.0020, 0, 0, 0])
    movel(p[new_pose[0], new_pose[1], new_pose[2], current_pose[3], current_pose[4], current_pose[5]], a=0.8, v=0.2000)
    report_progress()
    set_digital_out(0, True)
    new_pose = pose_trans(tuft_coords, p[0.4593, 0.7496, -0.0020, 0, 0, 0])
    movel(p[new_pose[0], new_pose[1], new_pose[2], current_pose[3], current_pose[4], current_pose[5]], a=1.2, v=0.0600)
    report_progress()
    set_digital_out(0, False)
    new_pose = pose_trans(tuft_coords, p[0.4593, 0.7496, 0.1500, 0, 0, 0])
    movel(p[new_pose[0], new_pose[1], new_pose[2], current_pose[3], current_pose[4], current_pose[5]], a=0.8, v=0.2000)
    report_progress()
    new_pose = pose_trans(tuft_coords, p[0.4612, 0.2984, 0.1500, 0, 0, 0])
    movel(p[new_pose[0], new_pose[1], new_pose[2], current_pose[3], current_pose[4], current_pose[5]], a=1.2, v=0.2000)
    report_progress()
    new_pose = pose_trans(tuft_coords, p[0.4612, 0.2984, -0.0020, 0, 0, 0])
    movel(p[new_pose[0], new_pose[1], new_pose[2], current_pose[3], current_pose[4], current_pose[5]], a=0.8, v=0.2000)
    report_progress()
    set_digital_out(0, True)
    new_pose = pose_trans(tuft_coords, p[0.4612, 0.7516, -0.0020, 0, 0, 0])
    movel(p[new_pose[0], new_pose[1], new_pose[2], current_pose[3], current_pose[4], current_pose[5]], a=1.2, v=0.0600)
    report_progress()
    set_digital_out(0, False)
    new_pose = pose_trans(tuft_coords, p[0.4612, 0.7516, 0.1500, 0, 0, 0])
    movel(p[new_pose[0], new_pose[1], new_pose[2], current_pose[3], current_pose[4], current_pose[5]], a=0.8, v=0.2000)
    report_progress()
    new_pose = pose_trans(tuft_coords, p[0.4632, 0.2964, 0.1500, 0, 0, 0])
    movel(p[new_pose[0], new_pose[1], new_pose[2], current_pose[3], current_pose[4], current_pose[5]], a=1.2, v=0.2000)
    report_progress()
    new_pose = pose_trans(tuft_coords, p[0.4632, 0.2964, -0.0020, 0, 0, 0])
    movel(p[new_pose[0], new_pose[1], new_pose[2], current_pose[3], current_pose[4], current_pose[5]], a=0.8, v=0.2000)
    report_progress()
    set_digital_out(0, True)
    new_pose = pose_trans(tuft_coords, p[0.4632, 0.7536, -0.0020, 0, 0, 0])
    movel(p[new_pose[0], new_pose[1], new_pose[2], current_pose[3], current_pose[4], current_pose[5]], a=1.2, v=0.0600)
    report_progress()
    set_digital_out(0, False)
    new_pose = pose_trans(tuft_coords, p[0.4632, 0.7536, 0.1500, 0, 0, 0])
    movel(p[new_pose[0], new_pose[1], new_pose[2], current_pose[3], current_pose[4], current_pose[5]], a=0.8, v=0.2000)
    report_progress()
    new_pose = pose_trans(tuft_coords, p[0.4651, 0.2944, 0.1500, 0, 0, 0])
    movel(p[new_pose[0], new_pose[1], new_pose[2], current_pose[3], current_pose[4], current_pose[5]], a=1.2, v=0.2000)
    report_progress()
    new_pose = pose_trans(tuft_coords, p[0.4651, 0.2944, -0.0020, 0, 0, 0])
    movel(p[new_pose[0], new_pose[1], new_pose[2], current_pose[3], current_pose[4], current_pose[5]], a=0.8, v=0.2000)
    report_progress()
    set_digital_out(0, True)
    new_pose = pose_trans(tuft_coords, p[0.4651, 0.7556, -0.0020, 0, 0, 0])
    movel(p[new_pose[0], new_pose[1], new_pose[2], current_pose[3], current_pose[4], current_pose[5]], a=1.2, v=0.0600)
    report_progress()
    set_digital_out(0, False)
    new_pose = pose_trans(tuft_coords, p[0.4651, 0.7556, 0.1500, 0, 0, 0])
    movel(p[new_pose[0], new_pose[1], new_pose[2], current_pose[3], current_pose[4], current_pose[5]], a=0.8, v=0.2000)
    report_progress()
    new_pose = pose_trans(tuft_coords, p[0.4671, 0.2905, 0.1500, 0, 0, 0])
    movel(p[new_pose[0], new_pose[1], new_pose[2], current_pose[3], current_pose[4], current_pose[5]], a=1.2, v=0.2000)
    report_progress()
    new_pose = pose_trans(tuft_coords, p[0.4671, 0.2905, -0.0020, 0, 0, 0])
    movel(p[new_pose[0], new_pose[1], new_pose[2], current_pose[3], current_pose[4], current_pose[5]], a=0.8, v=0.2000)
    report_progress()
    set_digital_out(0, True)
    new_pose = pose_trans(tuft_coords, p[0.4671, 0.7595, -0.0020, 0, 0, 0])
    movel(p[new_pose[0], new_pose[1], new_pose[2], current_pose[3], current_pose[4], current_pose[5]], a=1.2, v=0.0600)
    report_progress()
    set_digital_out(0, False)
    new_pose = pose_trans(tuft_coords, p[0.4671, 0.7595, 0.1500, 0, 0, 0])
    movel(p[new_pose[0], new_pose[1], new_pose[2], current_pose[3], current_pose[4], current_pose[5]], a=0.8, v=0.2000)
    report_progress()
    new_pose = pose_trans(tuft_coords, p[0.4690, 0.2885, 0.1500, 0, 0, 0])
    movel(p[new_pose[0], new_pose[1], new_pose[2], current_pose[3], current_pose[4], current_pose[5]], a=1.2, v=0.2000)
    report_progress()
    new_pose = pose_trans(tuft_coords, p[0.4690, 0.2885, -0.0020, 0, 0, 0])
    movel(p[new_pose[0], new_pose[1], new_pose[2], current_pose[3], current_pose[4], current_pose[5]], a=0.8, v=0.2000)
    report_progress()
    set_digital_out(0, True)
    new_pose = pose_trans(tuft_coords, p[0.4690, 0.7615, -0.0020, 0, 0, 0])
    movel(p[new_pose[0], new_pose[1], new_pose[2], current_pose[3], current_pose[4], current_pose[5]], a=1.2, v=0.0600)
    report_progress()
    set_digital_out(0, False)
    new_pose = pose_trans(tuft_coords, p[0.4690, 0.7615, 0.1500, 0, 0, 0])
    movel(p[new_pose[0], new_pose[1], new_pose[2], current_pose[3], current_pose[4], current_pose[5]], a=0.8, v=0.2000)
    report_progress()
    new_pose = pose_trans(tuft_coords, p[0.4710, 0.2865, 0.1500, 0, 0, 0])
    movel(p[new_pose[0], new_pose[1], new_pose[2], current_pose[3], current_pose[4], current_pose[5]], a=1.2, v=0.2000)
    report_progress()
    new_pose = pose_trans(tuft_coords, p[0.4710, 0.2865, -0.0020, 0, 0, 0])
    movel(p[new_pose[0], new_pose[1], new_pose[2], current_pose[3], current_pose[4], current_pose[5]], a=0.8, v=0.2000)
    report_progress()
    set_digital_out(0, True)
    new_pose = pose_trans(tuft_coords, p[0.4710, 0.7635, -0.0020, 0, 0, 0])
    movel(p[new_pose[0], new_pose[1], new_pose[2], current_pose[3], current_pose[4], current_pose[5]], a=1.2, v=0.0600)
    report_progress()
    set_digital_out(0, False)
    new_pose = pose_trans(tuft_coords, p[0.4710, 0.7635, 0.1500, 0, 0, 0])
    movel(p[new_pose[0], new_pose[1], new_pose[2], current_pose[3], current_pose[4], current_pose[5]], a=0.8, v=0.2000)
    report_progress()
    new_pose = pose_trans(tuft_coords, p[0.4729, 0.2845, 0.1500, 0, 0, 0])
    movel(p[new_pose[0], new_pose[1], new_pose[2], current_pose[3], current_pose[4], current_pose[5]], a=1.2, v=0.2000)
    report_progress()
    new_pose = pose_trans(tuft_coords, p[0.4729, 0.2845, -0.0020, 0, 0, 0])
    movel(p[new_pose[0], new_pose[1], new_pose[2], current_pose[3], current_pose[4], current_pose[5]], a=0.8, v=0.2000)
    report_progress()
    set_digital_out(0, True)
    new_pose = pose_trans(tuft_coords, p[0.4729, 0.7655, -0.0020, 0, 0, 0])
    movel(p[new_pose[0], new_pose[1], new_pose[2], current_pose[3], current_pose[4], current_pose[5]], a=1.2, v=0.0600)
    report_progress()
    set_digital_out(0, False)
    new_pose = pose_trans(tuft_coords, p[0.4729, 0.7655, 0.1500, 0, 0, 0])
    movel(p[new_pose[0], new_pose[1], new_pose[2], current_pose[3], current_pose[4], current_pose[5]], a=0.8, v=0.2000)
    report_progress()
    new_pose = pose_trans(tuft_coords, p[0.4749, 0.2826, 0.1500, 0, 0, 0])
    movel(p[new_pose[0], new_pose[1], new_pose[2], current_pose[3], current_pose[4], current_pose[5]], a=1.2, v=0.2000)
    report_progress()
    new_pose = pose_trans(tuft_coords, p[0.4749, 0.2826, -0.0020, 0, 0, 0])
    movel(p[new_pose[0], new_pose[1], new_pose[2], current_pose[3], current_pose[4], current_pose[5]], a=0.8, v=0.2000)
    report_progress()
    set_digital_out(0, True)
    new_pose = pose_trans(tuft_coords, p[0.4749, 0.7674, -0.0020, 0, 0, 0])
    movel(p[new_pose[0], new_pose[1], new_pose[2], current_pose[3], current_pose[4], current_pose[5]], a=1.2, v=0.0600)
    report_progress()
    set_digital_out(0, False)
    new_pose = pose_trans(tuft_coords, p[0.4749, 0.7674, 0.1500, 0, 0, 0])
    movel(p[new_pose[0], new_pose[1], new_pose[2], current_pose[3], current_pose[4], current_pose[5]], a=0.8, v=0.2000)
    report_progress()
    new_pose = pose_trans(tuft_coords, p[0.4768, 0.2786, 0.1500, 0, 0, 0])
    movel(p[new_pose[0], new_pose[1], new_pose[2], current_pose[3], current_pose[4], current_pose[5]], a=1.2, v=0.2000)
    report_progress()
    new_pose = pose_trans(tuft_coords, p[0.4768, 0.2786, -0.0020, 0, 0, 0])
    movel(p[new_pose[0], new_pose[1], new_pose[2], current_pose[3], current_pose[4], current_pose[5]], a=0.8, v=0.2000)
    report_progress()
    set_digital_out(0, True)
    new_pose = pose_trans(tuft_coords, p[0.4768, 0.7714, -0.0020, 0, 0, 0])
    movel(p[new_pose[0], new_pose[1], new_pose[2], current_pose[3], current_pose[4], current_pose[5]], a=1.2, v=0.0600)
    report_progress()
    set_digital_out(0, False)
    new_pose = pose_trans(tuft_coords, p[0.4768, 0.7714, 0.1500, 0, 0, 0])
    movel(p[new_pose[0], new_pose[1], new_pose[2], current_pose[3], current_pose[4], current_pose[5]], a=0.8, v=0.2000)
    report_progress()
    new_pose = pose_trans(tuft_coords, p[0.4788, 0.2766, 0.1500, 0, 0, 0])
    movel(p[new_pose[0], new_pose[1], new_pose[2], current_pose[3], current_pose[4], current_pose[5]], a=1.2, v=0.2000)
    report_progress()
    new_pose = pose_trans(tuft_coords, p[0.4788, 0.2766, -0.0020, 0, 0, 0])
    movel(p[new_pose[0], new_pose[1], new_pose[2], current_pose[3], current_pose[4], current_pose[5]], a=0.8, v=0.2000)
    report_progress()
    set_digital_out(0, True)
    new_pose = pose_trans(tuft_coords, p[0.4788, 0.7734, -0.0020, 0, 0, 0])
    movel(p[new_pose[0], new_pose[1], new_pose[2], current_pose[3], current_pose[4], current_pose[5]], a=1.2, v=0.0600)
    report_progress()
    set_digital_out(0, False)
    new_pose = pose_trans(tuft_coords, p[0.4788, 0.7734, 0.1500, 0, 0, 0])
    movel(p[new_pose[0], new_pose[1], new_pose[2], current_pose[3], current_pose[4], current_pose[5]], a=0.8, v=0.2000)
    report_progress()
    new_pose = pose_trans(tuft_coords, p[0.4807, 0.2746, 0.1500, 0, 0, 0])
    movel(p[new_pose[0], new_pose[1], new_pose[2], current_pose[3], current_pose[4], current_pose[5]], a=1.2, v=0.2000)
    report_progress()
    new_pose = pose_trans(tuft_coords, p[0.4807, 0.2746, -0.0020, 0, 0, 0])
    movel(p[new_pose[0], new_pose[1], new_pose[2], current_pose[3], current_pose[4], current_pose[5]], a=0.8, v=0.2000)
    report_progress()
    set_digital_out(0, True)
    new_pose = pose_trans(tuft_coords, p[0.4807, 0.7754, -0.0020, 0, 0, 0])
    movel(p[new_pose[0], new_pose[1], new_pose[2], current_pose[3], current_pose[4], current_pose[5]], a=1.2, v=0.0600)
    report_progress()
    set_digital_out(0, False)
    new_pose = pose_trans(tuft_coords, p[0.4807, 0.7754, 0.1500, 0, 0, 0])
    movel(p[new_pose[0], new_pose[1], new_pose[2], current_pose[3], current_pose[4], current_pose[5]], a=0.8, v=0.2000)
    report_progress()
    new_pose = pose_trans(tuft_coords, p[0.4826, 0.2727, 0.1500, 0, 0, 0])
    movel(p[new_pose[0], new_pose[1], new_pose[2], current_pose[3], current_pose[4], current_pose[5]], a=1.2, v=0.2000)
    report_progress()
    new_pose = pose_trans(tuft_coords, p[0.4826, 0.2727, -0.0020, 0, 0, 0])
    movel(p[new_pose[0], new_pose[1], new_pose[2], current_pose[3], current_pose[4], current_pose[5]], a=0.8, v=0.2000)
    report_progress()
    set_digital_out(0, True)
    new_pose = pose_trans(tuft_coords, p[0.4826, 0.7773, -0.0020, 0, 0, 0])
    movel(p[new_pose[0], new_pose[1], new_pose[2], current_pose[3], current_pose[4], current_pose[5]], a=1.2, v=0.0600)
    report_progress()
    set_digital_out(0, False)
    new_pose = pose_trans(tuft_coords, p[0.4826, 0.7773, 0.1500, 0, 0, 0])
    movel(p[new_pose[0], new_pose[1], new_pose[2], current_pose[3], current_pose[4], current_pose[5]], a=0.8, v=0.2000)
    report_progress()
    new_pose = pose_trans(tuft_coords, p[0.4846, 0.2707, 0.1500, 0, 0, 0])
    movel(p[new_pose[0], new_pose[1], new_pose[2], current_pose[3], current_pose[4], current_pose[5]], a=1.2, v=0.2000)
    report_progress()
    new_pose = pose_trans(tuft_coords, p[0.4846, 0.2707, -0.0020, 0, 0, 0])
    movel(p[new_pose[0], new_pose[1], new_pose[2], current_pose[3], current_pose[4], current_pose[5]], a=0.8, v=0.2000)
    report_progress()
    set_digital_out(0, True)
    new_pose = pose_trans(tuft_coords, p[0.4846, 0.7793, -0.0020, 0, 0, 0])
    movel(p[new_pose[0], new_pose[1], new_pose[2], current_pose[3], current_pose[4], current_pose[5]], a=1.2, v=0.0600)
    report_progress()
    set_digital_out(0, False)
    new_pose = pose_trans(tuft_coords, p[0.4846, 0.7793, 0.1500, 0, 0, 0])
    movel(p[new_pose[0], new_pose[1], new_pose[2], current_pose[3], current_pose[4], current_pose[5]], a=0.8, v=0.2000)
    report_progress()
    new_pose = pose_trans(tuft_coords, p[0.4865, 0.2687, 0.1500, 0, 0, 0])
    movel(p[new_pose[0], new_pose[1], new_pose[2], current_pose[3], current_pose[4], current_pose[5]], a=1.2, v=0.2000)
    report_progress()
    new_pose = pose_trans(tuft_coords, p[0.4865, 0.2687, -0.0020, 0, 0, 0])
    movel(p[new_pose[0], new_pose[1], new_pose[2], current_pose[3], current_pose[4], current_pose[5]], a=0.8, v=0.2000)
    report_progress()
    set_digital_out(0, True)
    new_pose = pose_trans(tuft_coords, p[0.4865, 0.7813, -0.0020, 0, 0, 0])
    movel(p[new_pose[0], new_pose[1], new_pose[2], current_pose[3], current_pose[4], current_pose[5]], a=1.2, v=0.0600)
    report_progress()
    set_digital_out(0, False)
    new_pose = pose_trans(tuft_coords, p[0.4865, 0.7813, 0.1500, 0, 0, 0])
    movel(p[new_pose[0], new_pose[1], new_pose[2], current_pose[3], current_pose[4], current_pose[5]], a=0.8, v=0.2000)
    report_progress()
    new_pose = pose_trans(tuft_coords, p[0.4885, 0.2667, 0.1500, 0, 0, 0])
    movel(p[new_pose[0], new_pose[1], new_pose[2], current_pose[3], current_pose[4], current_pose[5]], a=1.2, v=0.2000)
    report_progress()
    new_pose = pose_trans(tuft_coords, p[0.4885, 0.2667, -0.0020, 0, 0, 0])
    movel(p[new_pose[0], new_pose[1], new_pose[2], current_pose[3], current_pose[4], current_pose[5]], a=0.8, v=0.2000)
    report_progress()
    set_digital_out(0, True)
    new_pose = pose_trans(tuft_coords, p[0.4885, 0.7833, -0.0020, 0, 0, 0])
    movel(p[new_pose[0], new_pose[1], new_pose[2], current_pose[3], current_pose[4], current_pose[5]], a=1.2, v=0.0600)
    report_progress()
    set_digital_out(0, False)
    new_pose = pose_trans(tuft_coords, p[0.4885, 0.7833, 0.1500, 0, 0, 0])
    movel(p[new_pose[0], new_pose[1], new_pose[2], current_pose[3], current_pose[4], current_pose[5]], a=0.8, v=0.2000)
    report_progress()
    new_pose = pose_trans(tuft_coords, p[0.4904, 0.2647, 0.1500, 0, 0, 0])
    movel(p[new_pose[0], new_pose[1], new_pose[2], current_pose[3], current_pose[4], current_pose[5]], a=1.2, v=0.2000)
    report_progress()
    new_pose = pose_trans(tuft_coords, p[0.4904, 0.2647, -0.0020, 0, 0, 0])
    movel(p[new_pose[0], new_pose[1], new_pose[2], current_pose[3], current_pose[4], current_pose[5]], a=0.8, v=0.2000)
    report_progress()
    set_digital_out(0, True)
    new_pose = pose_trans(tuft_coords, p[0.4904, 0.7853, -0.0020, 0, 0, 0])
    movel(p[new_pose[0], new_pose[1], new_pose[2], current_pose[3], current_pose[4], current_pose[5]], a=1.2, v=0.0600)
    report_progress()
    set_digital_out(0, False)
    new_pose = pose_trans(tuft_coords, p[0.4904, 0.7853, 0.1500, 0, 0, 0])
    movel(p[new_pose[0], new_pose[1], new_pose[2], current_pose[3], current_pose[4], current_pose[5]], a=0.8, v=0.2000)
    report_progress()
    new_pose = pose_trans(tuft_coords, p[0.4924, 0.2628, 0.1500, 0, 0, 0])
    movel(p[new_pose[0], new_pose[1], new_pose[2], current_pose[3], current_pose[4], current_pose[5]], a=1.2, v=0.2000)
    report_progress()
    new_pose = pose_trans(tuft_coords, p[0.4924, 0.2628, -0.0020, 0, 0, 0])
    movel(p[new_pose[0], new_pose[1], new_pose[2], current_pose[3], current_pose[4], current_pose[5]], a=0.8, v=0.2000)
    report_progress()
    set_digital_out(0, True)
    new_pose = pose_trans(tuft_coords, p[0.4924, 0.7872, -0.0020, 0, 0, 0])
    movel(p[new_pose[0], new_pose[1], new_pose[2], current_pose[3], current_pose[4], current_pose[5]], a=1.2, v=0.0600)
    report_progress()
    set_digital_out(0, False)
    new_pose = pose_trans(tuft_coords, p[0.4924, 0.7872, 0.1500, 0, 0, 0])
    movel(p[new_pose[0], new_pose[1], new_pose[2], current_pose[3], current_pose[4], current_pose[5]], a=0.8, v=0.2000)
    report_progress()
    new_pose = pose_trans(tuft_coords, p[0.4943, 0.2608, 0.1500, 0, 0, 0])
    movel(p[new_pose[0], new_pose[1], new_pose[2], current_pose[3], current_pose[4], current_pose[5]], a=1.2, v=0.2000)
    report_progress()
    new_pose = pose_trans(tuft_coords, p[0.4943, 0.2608, -0.0020, 0, 0, 0])
    movel(p[new_pose[0], new_pose[1], new_pose[2], current_pose[3], current_pose[4], current_pose[5]], a=0.8, v=0.2000)
    report_progress()
    set_digital_out(0, True)
    new_pose = pose_trans(tuft_coords, p[0.4943, 0.7892, -0.0020, 0, 0, 0])
    movel(p[new_pose[0], new_pose[1], new_pose[2], current_pose[3], current_pose[4], current_pose[5]], a=1.2, v=0.0600)
    report_progress()
    set_digital_out(0, False)
    new_pose = pose_trans(tuft_coords, p[0.4943, 0.7892, 0.1500, 0, 0, 0])
    movel(p[new_pose[0], new_pose[1], new_pose[2], current_pose[3], current_pose[4], current_pose[5]], a=0.8, v=0.2000)
    report_progress()
    new_pose = pose_trans(tuft_coords, p[0.4963, 0.2588, 0.1500, 0, 0, 0])
    movel(p[new_pose[0], new_pose[1], new_pose[2], current_pose[3], current_pose[4], current_pose[5]], a=1.2, v=0.2000)
    report_progress()
    new_pose = pose_trans(tuft_coords, p[0.4963, 0.2588, -0.0020, 0, 0, 0])
    movel(p[new_pose[0], new_pose[1], new_pose[2], current_pose[3], current_pose[4], current_pose[5]], a=0.8, v=0.2000)
    report_progress()
    set_digital_out(0, True)
    new_pose = pose_trans(tuft_coords, p[0.4963, 0.7912, -0.0020, 0, 0, 0])
    movel(p[new_pose[0], new_pose[1], new_pose[2], current_pose[3], current_pose[4], current_pose[5]], a=1.2, v=0.0600)
    report_progress()
    set_digital_out(0, False)
    new_pose = pose_trans(tuft_coords, p[0.4963, 0.7912, 0.1500, 0, 0, 0])
    movel(p[new_pose[0], new_pose[1], new_pose[2], current_pose[3], current_pose[4], current_pose[5]], a=0.8, v=0.2000)
    report_progress()
    new_pose = pose_trans(tuft_coords, p[0.4982, 0.2568, 0.1500, 0, 0, 0])
    movel(p[new_pose[0], new_pose[1], new_pose[2], current_pose[3], current_pose[4], current_pose[5]], a=1.2, v=0.2000)
    report_progress()
    new_pose = pose_trans(tuft_coords, p[0.4982, 0.2568, -0.0020, 0, 0, 0])
    movel(p[new_pose[0], new_pose[1], new_pose[2], current_pose[3], current_pose[4], current_pose[5]], a=0.8, v=0.2000)
    report_progress()
    set_digital_out(0, True)
    new_pose = pose_trans(tuft_coords, p[0.4982, 0.7932, -0.0020, 0, 0, 0])
    movel(p[new_pose[0], new_pose[1], new_pose[2], current_pose[3], current_pose[4], current_pose[5]], a=1.2, v=0.0600)
    report_progress()
    set_digital_out(0, False)
    new_pose = pose_trans(tuft_coords, p[0.4982, 0.7932, 0.1500, 0, 0, 0])
    movel(p[new_pose[0], new_pose[1], new_pose[2], current_pose[3], current_pose[4], current_pose[5]], a=0.8, v=0.2000)
    report_progress()
    new_pose = pose_trans(tuft_coords, p[0.5001, 0.2548, 0.1500, 0, 0, 0])
    movel(p[new_pose[0], new_pose[1], new_pose[2], current_pose[3], current_pose[4], current_pose[5]], a=1.2, v=0.2000)
    report_progress()
    new_pose = pose_trans(tuft_coords, p[0.5001, 0.2548, -0.0020, 0, 0, 0])
    movel(p[new_pose[0], new_pose[1], new_pose[2], current_pose[3], current_pose[4], current_pose[5]], a=0.8, v=0.2000)
    report_progress()
    set_digital_out(0, True)
    new_pose = pose_trans(tuft_coords, p[0.5001, 0.7952, -0.0020, 0, 0, 0])
    movel(p[new_pose[0], new_pose[1], new_pose[2], current_pose[3], current_pose[4], current_pose[5]], a=1.2, v=0.0600)
    report_progress()
    set_digital_out(0, False)
    new_pose = pose_trans(tuft_coords, p[0.5001, 0.7952, 0.1500, 0, 0, 0])
    movel(p[new_pose[0], new_pose[1], new_pose[2], current_pose[3], current_pose[4], current_pose[5]], a=0.8, v=0.2000)
    report_progress()
    new_pose = pose_trans(tuft_coords, p[0.5021, 0.2529, 0.1500, 0, 0, 0])
    movel(p[new_pose[0], new_pose[1], new_pose[2], current_pose[3], current_pose[4], current_pose[5]], a=1.2, v=0.2000)
    report_progress()
    new_pose = pose_trans(tuft_coords, p[0.5021, 0.2529, -0.0020, 0, 0, 0])
    movel(p[new_pose[0], new_pose[1], new_pose[2], current_pose[3], current_pose[4], current_pose[5]], a=0.8, v=0.2000)
    report_progress()
    set_digital_out(0, True)
    new_pose = pose_trans(tuft_coords, p[0.5021, 0.7971, -0.0020, 0, 0, 0])
    movel(p[new_pose[0], new_pose[1], new_pose[2], current_pose[3], current_pose[4], current_pose[5]], a=1.2, v=0.0600)
    report_progress()
    set_digital_out(0, False)
    new_pose = pose_trans(tuft_coords, p[0.5021, 0.7971, 0.1500, 0, 0, 0])
    movel(p[new_pose[0], new_pose[1], new_pose[2], current_pose[3], current_pose[4], current_pose[5]], a=0.8, v=0.2000)
    report_progress()
    new_pose = pose_trans(tuft_coords, p[0.5040, 0.2509, 0.1500, 0, 0, 0])
    movel(p[new_pose[0], new_pose[1], new_pose[2], current_pose[3], current_pose[4], current_pose[5]], a=1.2, v=0.2000)
    report_progress()
    new_pose = pose_trans(tuft_coords, p[0.5040, 0.2509, -0.0020, 0, 0, 0])
    movel(p[new_pose[0], new_pose[1], new_pose[2], current_pose[3], current_pose[4], current_pose[5]], a=0.8, v=0.2000)
    report_progress()
    set_digital_out(0, True)
    new_pose = pose_trans(tuft_coords, p[0.5040, 0.7991, -0.0020, 0, 0, 0])
    movel(p[new_pose[0], new_pose[1], new_pose[2], current_pose[3], current_pose[4], current_pose[5]], a=1.2, v=0.0600)
    report_progress()
    set_digital_out(0, False)
    new_pose = pose_trans(tuft_coords, p[0.5040, 0.7991, 0.1500, 0, 0, 0])
    movel(p[new_pose[0], new_pose[1], new_pose[2], current_pose[3], current_pose[4], current_pose[5]], a=0.8, v=0.2000)
    report_progress()
    new_pose = pose_trans(tuft_coords, p[0.5060, 0.2489, 0.1500, 0, 0, 0])
    movel(p[new_pose[0], new_pose[1], new_pose[2], current_pose[3], current_pose[4], current_pose[5]], a=1.2, v=0.2000)
    report_progress()
    new_pose = pose_trans(tuft_coords, p[0.5060, 0.2489, -0.0020, 0, 0, 0])
    movel(p[new_pose[0], new_pose[1], new_pose[2], current_pose[3], current_pose[4], current_pose[5]], a=0.8, v=0.2000)
    report_progress()
    set_digital_out(0, True)
    new_pose = pose_trans(tuft_coords, p[0.5060, 0.8011, -0.0020, 0, 0, 0])
    movel(p[new_pose[0], new_pose[1], new_pose[2], current_pose[3], current_pose[4], current_pose[5]], a=1.2, v=0.0600)
    report_progress()
    set_digital_out(0, False)
    new_pose = pose_trans(tuft_coords, p[0.5060, 0.8011, 0.1500, 0, 0, 0])
    movel(p[new_pose[0], new_pose[1], new_pose[2], current_pose[3], current_pose[4], current_pose[5]], a=0.8, v=0.2000)
    report_progress()
    new_pose = pose_trans(tuft_coords, p[0.5079, 0.2469, 0.1500, 0, 0, 0])
    movel(p[new_pose[0], new_pose[1], new_pose[2], current_pose[3], current_pose[4], current_pose[5]], a=1.2, v=0.2000)
    report_progress()
    new_pose = pose_trans(tuft_coords, p[0.5079, 0.2469, -0.0020, 0, 0, 0])
    movel(p[new_pose[0], new_pose[1], new_pose[2], current_pose[3], current_pose[4], current_pose[5]], a=0.8, v=0.2000)
    report_progress()
    set_digital_out(0, True)
    new_pose = pose_trans(tuft_coords, p[0.5079, 0.8031, -0.0020, 0, 0, 0])
    movel(p[new_pose[0], new_pose[1], new_pose[2], current_pose[3], current_pose[4], current_pose[5]], a=1.2, v=0.0600)
    report_progress()
    set_digital_out(0, False)
    new_pose = pose_trans(tuft_coords, p[0.5079, 0.8031, 0.1500, 0, 0, 0])
    movel(p[new_pose[0], new_pose[1], new_pose[2], current_pose[3], current_pose[4], current_pose[5]], a=0.8, v=0.2000)
    report_progress()
    new_pose = pose_trans(tuft_coords, p[0.5099, 0.2469, 0.1500, 0, 0, 0])
    movel(p[new_pose[0], new_pose[1], new_pose[2], current_pose[3], current_pose[4], current_pose[5]], a=1.2, v=0.2000)
    report_progress()
    new_pose = pose_trans(tuft_coords, p[0.5099, 0.2469, -0.0020, 0, 0, 0])
    movel(p[new_pose[0], new_pose[1], new_pose[2], current_pose[3], current_pose[4], current_pose[5]], a=0.8, v=0.2000)
    report_progress()
    set_digital_out(0, True)
    new_pose = pose_trans(tuft_coords, p[0.5099, 0.8031, -0.0020, 0, 0, 0])
    movel(p[new_pose[0], new_pose[1], new_pose[2], current_pose[3], current_pose[4], current_pose[5]], a=1.2, v=0.0600)
    report_progress()
    set_digital_out(0, False)
    new_pose = pose_trans(tuft_coords, p[0.5099, 0.8031, 0.1500, 0, 0, 0])
    movel(p[new_pose[0], new_pose[1], new_pose[2], current_pose[3], current_pose[4], current_pose[5]], a=0.8, v=0.2000)
    report_progress()
    new_pose = pose_trans(tuft_coords, p[0.5118, 0.2449, 0.1500, 0, 0, 0])
    movel(p[new_pose[0], new_pose[1], new_pose[2], current_pose[3], current_pose[4], current_pose[5]], a=1.2, v=0.2000)
    report_progress()
    new_pose = pose_trans(tuft_coords, p[0.5118, 0.2449, -0.0020, 0, 0, 0])
    movel(p[new_pose[0], new_pose[1], new_pose[2], current_pose[3], current_pose[4], current_pose[5]], a=0.8, v=0.2000)
    report_progress()
    set_digital_out(0, True)
    new_pose = pose_trans(tuft_coords, p[0.5118, 0.8051, -0.0020, 0, 0, 0])
    movel(p[new_pose[0], new_pose[1], new_pose[2], current_pose[3], current_pose[4], current_pose[5]], a=1.2, v=0.0600)
    report_progress()
    set_digital_out(0, False)
    new_pose = pose_trans(tuft_coords, p[0.5118, 0.8051, 0.1500, 0, 0, 0])
    movel(p[new_pose[0], new_pose[1], new_pose[2], current_pose[3], current_pose[4], current_pose[5]], a=0.8, v=0.2000)
    report_progress()
    new_pose = pose_trans(tuft_coords, p[0.5138, 0.2430, 0.1500, 0, 0, 0])
    movel(p[new_pose[0], new_pose[1], new_pose[2], current_pose[3], current_pose[4], current_pose[5]], a=1.2, v=0.2000)
    report_progress()
    new_pose = pose_trans(tuft_coords, p[0.5138, 0.2430, -0.0020, 0, 0, 0])
    movel(p[new_pose[0], new_pose[1], new_pose[2], current_pose[3], current_pose[4], current_pose[5]], a=0.8, v=0.2000)
    report_progress()
    set_digital_out(0, True)
    new_pose = pose_trans(tuft_coords, p[0.5138, 0.8070, -0.0020, 0, 0, 0])
    movel(p[new_pose[0], new_pose[1], new_pose[2], current_pose[3], current_pose[4], current_pose[5]], a=1.2, v=0.0600)
    report_progress()
    set_digital_out(0, False)
    new_pose = pose_trans(tuft_coords, p[0.5138, 0.8070, 0.1500, 0, 0, 0])
    movel(p[new_pose[0], new_pose[1], new_pose[2], current_pose[3], current_pose[4], current_pose[5]], a=0.8, v=0.2000)
    report_progress()
    new_pose = pose_trans(tuft_coords, p[0.5157, 0.2410, 0.1500, 0, 0, 0])
    movel(p[new_pose[0], new_pose[1], new_pose[2], current_pose[3], current_pose[4], current_pose[5]], a=1.2, v=0.2000)
    report_progress()
    new_pose = pose_trans(tuft_coords, p[0.5157, 0.2410, -0.0020, 0, 0, 0])
    movel(p[new_pose[0], new_pose[1], new_pose[2], current_pose[3], current_pose[4], current_pose[5]], a=0.8, v=0.2000)
    report_progress()
    set_digital_out(0, True)
    new_pose = pose_trans(tuft_coords, p[0.5157, 0.8090, -0.0020, 0, 0, 0])
    movel(p[new_pose[0], new_pose[1], new_pose[2], current_pose[3], current_pose[4], current_pose[5]], a=1.2, v=0.0600)
    report_progress()
    set_digital_out(0, False)
    new_pose = pose_trans(tuft_coords, p[0.5157, 0.8090, 0.1500, 0, 0, 0])
    movel(p[new_pose[0], new_pose[1], new_pose[2], current_pose[3], current_pose[4], current_pose[5]], a=0.8, v=0.2000)
    report_progress()
    new_pose = pose_trans(tuft_coords, p[0.5176, 0.2390, 0.1500, 0, 0, 0])
    movel(p[new_pose[0], new_pose[1], new_pose[2], current_pose[3], current_pose[4], current_pose[5]], a=1.2, v=0.2000)
    report_progress()
    new_pose = pose_trans(tuft_coords, p[0.5176, 0.2390, -0.0020, 0, 0, 0])
    movel(p[new_pose[0], new_pose[1], new_pose[2], current_pose[3], current_pose[4], current_pose[5]], a=0.8, v=0.2000)
    report_progress()
    set_digital_out(0, True)
    new_pose = pose_trans(tuft_coords, p[0.5176, 0.8110, -0.0020, 0, 0, 0])
    movel(p[new_pose[0], new_pose[1], new_pose[2], current_pose[3], current_pose[4], current_pose[5]], a=1.2, v=0.0600)
    report_progress()
    set_digital_out(0, False)
    new_pose = pose_trans(tuft_coords, p[0.5176, 0.8110, 0.1500, 0, 0, 0])
    movel(p[new_pose[0], new_pose[1], new_pose[2], current_pose[3], current_pose[4], current_pose[5]], a=0.8, v=0.2000)
    report_progress()
    new_pose = pose_trans(tuft_coords, p[0.5196, 0.2370, 0.1500, 0, 0, 0])
    movel(p[new_pose[0], new_pose[1], new_pose[2], current_pose[3], current_pose[4], current_pose[5]], a=1.2, v=0.2000)
    report_progress()
    new_pose = pose_trans(tuft_coords, p[0.5196, 0.2370, -0.0020, 0, 0, 0])
    movel(p[new_pose[0], new_pose[1], new_pose[2], current_pose[3], current_pose[4], current_pose[5]], a=0.8, v=0.2000)
    report_progress()
    set_digital_out(0, True)
    new_pose = pose_trans(tuft_coords, p[0.5196, 0.8130, -0.0020, 0, 0, 0])
    movel(p[new_pose[0], new_pose[1], new_pose[2], current_pose[3], current_pose[4], current_pose[5]], a=1.2, v=0.0600)
    report_progress()
    set_digital_out(0, False)
    new_pose = pose_trans(tuft_coords, p[0.5196, 0.8130, 0.1500, 0, 0, 0])
    movel(p[new_pose[0], new_pose[1], new_pose[2], current_pose[3], current_pose[4], current_pose[5]], a=0.8, v=0.2000)
    report_progress()
    new_pose = pose_trans(tuft_coords, p[0.5215, 0.2351, 0.1500, 0, 0, 0])
    movel(p[new_pose[0], new_pose[1], new_pose[2], current_pose[3], current_pose[4], current_pose[5]], a=1.2, v=0.2000)
    report_progress()
    new_pose = pose_trans(tuft_coords, p[0.5215, 0.2351, -0.0020, 0, 0, 0])
    movel(p[new_pose[0], new_pose[1], new_pose[2], current_pose[3], current_pose[4], current_pose[5]], a=0.8, v=0.2000)
    report_progress()
    set_digital_out(0, True)
    new_pose = pose_trans(tuft_coords, p[0.5215, 0.8149, -0.0020, 0, 0, 0])
    movel(p[new_pose[0], new_pose[1], new_pose[2], current_pose[3], current_pose[4], current_pose[5]], a=1.2, v=0.0600)
    report_progress()
    set_digital_out(0, False)
    new_pose = pose_trans(tuft_coords, p[0.5215, 0.8149, 0.1500, 0, 0, 0])
    movel(p[new_pose[0], new_pose[1], new_pose[2], current_pose[3], current_pose[4], current_pose[5]], a=0.8, v=0.2000)
    report_progress()
    new_pose = pose_trans(tuft_coords, p[0.5235, 0.2351, 0.1500, 0, 0, 0])
    movel(p[new_pose[0], new_pose[1], new_pose[2], current_pose[3], current_pose[4], current_pose[5]], a=1.2, v=0.2000)
    report_progress()
    new_pose = pose_trans(tuft_coords, p[0.5235, 0.2351, -0.0020, 0, 0, 0])
    movel(p[new_pose[0], new_pose[1], new_pose[2], current_pose[3], current_pose[4], current_pose[5]], a=0.8, v=0.2000)
    report_progress()
    set_digital_out(0, True)
    new_pose = pose_trans(tuft_coords, p[0.5235, 0.8149, -0.0020, 0, 0, 0])
    movel(p[new_pose[0], new_pose[1], new_pose[2], current_pose[3], current_pose[4], current_pose[5]], a=1.2, v=0.0600)
    report_progress()
    set_digital_out(0, False)
    new_pose = pose_trans(tuft_coords, p[0.5235, 0.8149, 0.1500, 0, 0, 0])
    movel(p[new_pose[0], new_pose[1], new_pose[2], current_pose[3], current_pose[4], current_pose[5]], a=0.8, v=0.2000)
    report_progress()
    new_pose = pose_trans(tuft_coords, p[0.5254, 0.2331, 0.1500, 0, 0, 0])
    movel(p[new_pose[0], new_pose[1], new_pose[2], current_pose[3], current_pose[4], current_pose[5]], a=1.2, v=0.2000)
    report_progress()
    new_pose = pose_trans(tuft_coords, p[0.5254, 0.2331, -0.0020, 0, 0, 0])
    movel(p[new_pose[0], new_pose[1], new_pose[2], current_pose[3], current_pose[4], current_pose[5]], a=0.8, v=0.2000)
    report_progress()
    set_digital_out(0, True)
    new_pose = pose_trans(tuft_coords, p[0.5254, 0.8169, -0.0020, 0, 0, 0])
    movel(p[new_pose[0], new_pose[1], new_pose[2], current_pose[3], current_pose[4], current_pose[5]], a=1.2, v=0.0600)
    report_progress()
    set_digital_out(0, False)
    new_pose = pose_trans(tuft_coords, p[0.5254, 0.8169, 0.1500, 0, 0, 0])
    movel(p[new_pose[0], new_pose[1], new_pose[2], current_pose[3], current_pose[4], current_pose[5]], a=0.8, v=0.2000)
    report_progress()
    new_pose = pose_trans(tuft_coords, p[0.5274, 0.2311, 0.1500, 0, 0, 0])
    movel(p[new_pose[0], new_pose[1], new_pose[2], current_pose[3], current_pose[4], current_pose[5]], a=1.2, v=0.2000)
    report_progress()
    new_pose = pose_trans(tuft_coords, p[0.5274, 0.2311, -0.0020, 0, 0, 0])
    movel(p[new_pose[0], new_pose[1], new_pose[2], current_pose[3], current_pose[4], current_pose[5]], a=0.8, v=0.2000)
    report_progress()
    set_digital_out(0, True)
    new_pose = pose_trans(tuft_coords, p[0.5274, 0.8189, -0.0020, 0, 0, 0])
    movel(p[new_pose[0], new_pose[1], new_pose[2], current_pose[3], current_pose[4], current_pose[5]], a=1.2, v=0.0600)
    report_progress()
    set_digital_out(0, False)
    new_pose = pose_trans(tuft_coords, p[0.5274, 0.8189, 0.1500, 0, 0, 0])
    movel(p[new_pose[0], new_pose[1], new_pose[2], current_pose[3], current_pose[4], current_pose[5]], a=0.8, v=0.2000)
    report_progress()
    new_pose = pose_trans(tuft_coords, p[0.5293, 0.2291, 0.1500, 0, 0, 0])
    movel(p[new_pose[0], new_pose[1], new_pose[2], current_pose[3], current_pose[4], current_pose[5]], a=1.2, v=0.2000)
    report_progress()
    new_pose = pose_trans(tuft_coords, p[0.5293, 0.2291, -0.0020, 0, 0, 0])
    movel(p[new_pose[0], new_pose[1], new_pose[2], current_pose[3], current_pose[4], current_pose[5]], a=0.8, v=0.2000)
    report_progress()
    set_digital_out(0, True)
    new_pose = pose_trans(tuft_coords, p[0.5293, 0.8209, -0.0020, 0, 0, 0])
    movel(p[new_pose[0], new_pose[1], new_pose[2], current_pose[3], current_pose[4], current_pose[5]], a=1.2, v=0.0600)
    report_progress()
    set_digital_out(0, False)
    new_pose = pose_trans(tuft_coords, p[0.5293, 0.8209, 0.1500, 0, 0, 0])
    movel(p[new_pose[0], new_pose[1], new_pose[2], current_pose[3], current_pose[4], current_pose[5]], a=0.8, v=0.2000)
    report_progress()
    new_pose = pose_trans(tuft_coords, p[0.5313, 0.2291, 0.1500, 0, 0, 0])
    movel(p[new_pose[0], new_pose[1], new_pose[2], current_pose[3], current_pose[4], current_pose[5]], a=1.2, v=0.2000)
    report_progress()
    new_pose = pose_trans(tuft_coords, p[0.5313, 0.2291, -0.0020, 0, 0, 0])
    movel(p[new_pose[0], new_pose[1], new_pose[2], current_pose[3], current_pose[4], current_pose[5]], a=0.8, v=0.2000)
    report_progress()
    set_digital_out(0, True)
    new_pose = pose_trans(tuft_coords, p[0.5313, 0.8209, -0.0020, 0, 0, 0])
    movel(p[new_pose[0], new_pose[1], new_pose[2], current_pose[3], current_pose[4], current_pose[5]], a=1.2, v=0.0600)
    report_progress()
    set_digital_out(0, False)
    new_pose = pose_trans(tuft_coords, p[0.5313, 0.8209, 0.1500, 0, 0, 0])
    movel(p[new_pose[0], new_pose[1], new_pose[2], current_pose[3], current_pose[4], current_pose[5]], a=0.8, v=0.2000)
    report_progress()
    new_pose = pose_trans(tuft_coords, p[0.5332, 0.2271, 0.1500, 0, 0, 0])
    movel(p[new_pose[0], new_pose[1], new_pose[2], current_pose[3], current_pose[4], current_pose[5]], a=1.2, v=0.2000)
    report_progress()
    new_pose = pose_trans(tuft_coords, p[0.5332, 0.2271, -0.0020, 0, 0, 0])
    movel(p[new_pose[0], new_pose[1], new_pose[2], current_pose[3], current_pose[4], current_pose[5]], a=0.8, v=0.2000)
    report_progress()
    set_digital_out(0, True)
    new_pose = pose_trans(tuft_coords, p[0.5332, 0.8229, -0.0020, 0, 0, 0])
    movel(p[new_pose[0], new_pose[1], new_pose[2], current_pose[3], current_pose[4], current_pose[5]], a=1.2, v=0.0600)
    report_progress()
    set_digital_out(0, False)
    new_pose = pose_trans(tuft_coords, p[0.5332, 0.8229, 0.1500, 0, 0, 0])
    movel(p[new_pose[0], new_pose[1], new_pose[2], current_pose[3], current_pose[4], current_pose[5]], a=0.8, v=0.2000)
    report_progress()
    new_pose = pose_trans(tuft_coords, p[0.5351, 0.2252, 0.1500, 0, 0, 0])
    movel(p[new_pose[0], new_pose[1], new_pose[2], current_pose[3], current_pose[4], current_pose[5]], a=1.2, v=0.2000)
    report_progress()
    new_pose = pose_trans(tuft_coords, p[0.5351, 0.2252, -0.0020, 0, 0, 0])
    movel(p[new_pose[0], new_pose[1], new_pose[2], current_pose[3], current_pose[4], current_pose[5]], a=0.8, v=0.2000)
    report_progress()
    set_digital_out(0, True)
    new_pose = pose_trans(tuft_coords, p[0.5351, 0.8248, -0.0020, 0, 0, 0])
    movel(p[new_pose[0], new_pose[1], new_pose[2], current_pose[3], current_pose[4], current_pose[5]], a=1.2, v=0.0600)
    report_progress()
    set_digital_out(0, False)
    new_pose = pose_trans(tuft_coords, p[0.5351, 0.8248, 0.1500, 0, 0, 0])
    movel(p[new_pose[0], new_pose[1], new_pose[2], current_pose[3], current_pose[4], current_pose[5]], a=0.8, v=0.2000)
    report_progress()
    new_pose = pose_trans(tuft_coords, p[0.5371, 0.2232, 0.1500, 0, 0, 0])
    movel(p[new_pose[0], new_pose[1], new_pose[2], current_pose[3], current_pose[4], current_pose[5]], a=1.2, v=0.2000)
    report_progress()
    new_pose = pose_trans(tuft_coords, p[0.5371, 0.2232, -0.0020, 0, 0, 0])
    movel(p[new_pose[0], new_pose[1], new_pose[2], current_pose[3], current_pose[4], current_pose[5]], a=0.8, v=0.2000)
    report_progress()
    set_digital_out(0, True)
    new_pose = pose_trans(tuft_coords, p[0.5371, 0.8268, -0.0020, 0, 0, 0])
    movel(p[new_pose[0], new_pose[1], new_pose[2], current_pose[3], current_pose[4], current_pose[5]], a=1.2, v=0.0600)
    report_progress()
    set_digital_out(0, False)
    new_pose = pose_trans(tuft_coords, p[0.5371, 0.8268, 0.1500, 0, 0, 0])
    movel(p[new_pose[0], new_pose[1], new_pose[2], current_pose[3], current_pose[4], current_pose[5]], a=0.8, v=0.2000)
    report_progress()
    new_pose = pose_trans(tuft_coords, p[0.5390, 0.2232, 0.1500, 0, 0, 0])
    movel(p[new_pose[0], new_pose[1], new_pose[2], current_pose[3], current_pose[4], current_pose[5]], a=1.2, v=0.2000)
    report_progress()
    new_pose = pose_trans(tuft_coords, p[0.5390, 0.2232, -0.0020, 0, 0, 0])
    movel(p[new_pose[0], new_pose[1], new_pose[2], current_pose[3], current_pose[4], current_pose[5]], a=0.8, v=0.2000)
    report_progress()
    set_digital_out(0, True)
    new_pose = pose_trans(tuft_coords, p[0.5390, 0.8268, -0.0020, 0, 0, 0])
    movel(p[new_pose[0], new_pose[1], new_pose[2], current_pose[3], current_pose[4], current_pose[5]], a=1.2, v=0.0600)
    report_progress()
    set_digital_out(0, False)
    new_pose = pose_trans(tuft_coords, p[0.5390, 0.8268, 0.1500, 0, 0, 0])
    movel(p[new_pose[0], new_pose[1], new_pose[2], current_pose[3], current_pose[4], current_pose[5]], a=0.8, v=0.2000)
    report_progress()
    new_pose = pose_trans(tuft_coords, p[0.5410, 0.2212, 0.1500, 0, 0, 0])
    movel(p[new_pose[0], new_pose[1], new_pose[2], current_pose[3], current_pose[4], current_pose[5]], a=1.2, v=0.2000)
    report_progress()
    new_pose = pose_trans(tuft_coords, p[0.5410, 0.2212, -0.0020, 0, 0, 0])
    movel(p[new_pose[0], new_pose[1], new_pose[2], current_pose[3], current_pose[4], current_pose[5]], a=0.8, v=0.2000)
    report_progress()
    set_digital_out(0, True)
    new_pose = pose_trans(tuft_coords, p[0.5410, 0.8288, -0.0020, 0, 0, 0])
    movel(p[new_pose[0], new_pose[1], new_pose[2], current_pose[3], current_pose[4], current_pose[5]], a=1.2, v=0.0600)
    report_progress()
    set_digital_out(0, False)
    new_pose = pose_trans(tuft_coords, p[0.5410, 0.8288, 0.1500, 0, 0, 0])
    movel(p[new_pose[0], new_pose[1], new_pose[2], current_pose[3], current_pose[4], current_pose[5]], a=0.8, v=0.2000)
    report_progress()
    new_pose = pose_trans(tuft_coords, p[0.5429, 0.2192, 0.1500, 0, 0, 0])
    movel(p[new_pose[0], new_pose[1], new_pose[2], current_pose[3], current_pose[4], current_pose[5]], a=1.2, v=0.2000)
    report_progress()
    new_pose = pose_trans(tuft_coords, p[0.5429, 0.2192, -0.0020, 0, 0, 0])
    movel(p[new_pose[0], new_pose[1], new_pose[2], current_pose[3], current_pose[4], current_pose[5]], a=0.8, v=0.2000)
    report_progress()
    set_digital_out(0, True)
    new_pose = pose_trans(tuft_coords, p[0.5429, 0.8308, -0.0020, 0, 0, 0])
    movel(p[new_pose[0], new_pose[1], new_pose[2], current_pose[3], current_pose[4], current_pose[5]], a=1.2, v=0.0600)
    report_progress()
    set_digital_out(0, False)
    new_pose = pose_trans(tuft_coords, p[0.5429, 0.8308, 0.1500, 0, 0, 0])
    movel(p[new_pose[0], new_pose[1], new_pose[2], current_pose[3], current_pose[4], current_pose[5]], a=0.8, v=0.2000)
    report_progress()
    new_pose = pose_trans(tuft_coords, p[0.5449, 0.2192, 0.1500, 0, 0, 0])
    movel(p[new_pose[0], new_pose[1], new_pose[2], current_pose[3], current_pose[4], current_pose[5]], a=1.2, v=0.2000)
    report_progress()
    new_pose = pose_trans(tuft_coords, p[0.5449, 0.2192, -0.0020, 0, 0, 0])
    movel(p[new_pose[0], new_pose[1], new_pose[2], current_pose[3], current_pose[4], current_pose[5]], a=0.8, v=0.2000)
    report_progress()
    set_digital_out(0, True)
    new_pose = pose_trans(tuft_coords, p[0.5449, 0.8308, -0.0020, 0, 0, 0])
    movel(p[new_pose[0], new_pose[1], new_pose[2], current_pose[3], current_pose[4], current_pose[5]], a=1.2, v=0.0600)
    report_progress()
    set_digital_out(0, False)
    new_pose = pose_trans(tuft_coords, p[0.5449, 0.8308, 0.1500, 0, 0, 0])
    movel(p[new_pose[0], new_pose[1], new_pose[2], current_pose[3], current_pose[4], current_pose[5]], a=0.8, v=0.2000)
    report_progress()
    new_pose = pose_trans(tuft_coords, p[0.5468, 0.2172, 0.1500, 0, 0, 0])
    movel(p[new_pose[0], new_pose[1], new_pose[2], current_pose[3], current_pose[4], current_pose[5]], a=1.2, v=0.2000)
    report_progress()
    new_pose = pose_trans(tuft_coords, p[0.5468, 0.2172, -0.0020, 0, 0, 0])
    movel(p[new_pose[0], new_pose[1], new_pose[2], current_pose[3], current_pose[4], current_pose[5]], a=0.8, v=0.2000)
    report_progress()
    set_digital_out(0, True)
    new_pose = pose_trans(tuft_coords, p[0.5468, 0.8328, -0.0020, 0, 0, 0])
    movel(p[new_pose[0], new_pose[1], new_pose[2], current_pose[3], current_pose[4], current_pose[5]], a=1.2, v=0.0600)
    report_progress()
    set_digital_out(0, False)
    new_pose = pose_trans(tuft_coords, p[0.5468, 0.8328, 0.1500, 0, 0, 0])
    movel(p[new_pose[0], new_pose[1], new_pose[2], current_pose[3], current_pose[4], current_pose[5]], a=0.8, v=0.2000)
    report_progress()
    new_pose = pose_trans(tuft_coords, p[0.5487, 0.2153, 0.1500, 0, 0, 0])
    movel(p[new_pose[0], new_pose[1], new_pose[2], current_pose[3], current_pose[4], current_pose[5]], a=1.2, v=0.2000)
    report_progress()
    new_pose = pose_trans(tuft_coords, p[0.5487, 0.2153, -0.0020, 0, 0, 0])
    movel(p[new_pose[0], new_pose[1], new_pose[2], current_pose[3], current_pose[4], current_pose[5]], a=0.8, v=0.2000)
    report_progress()
    set_digital_out(0, True)
    new_pose = pose_trans(tuft_coords, p[0.5487, 0.8347, -0.0020, 0, 0, 0])
    movel(p[new_pose[0], new_pose[1], new_pose[2], current_pose[3], current_pose[4], current_pose[5]], a=1.2, v=0.0600)
    report_progress()
    set_digital_out(0, False)
    new_pose = pose_trans(tuft_coords, p[0.5487, 0.8347, 0.1500, 0, 0, 0])
    movel(p[new_pose[0], new_pose[1], new_pose[2], current_pose[3], current_pose[4], current_pose[5]], a=0.8, v=0.2000)
    report_progress()
    new_pose = pose_trans(tuft_coords, p[0.5507, 0.2153, 0.1500, 0, 0, 0])
    movel(p[new_pose[0], new_pose[1], new_pose[2], current_pose[3], current_pose[4], current_pose[5]], a=1.2, v=0.2000)
    report_progress()
    new_pose = pose_trans(tuft_coords, p[0.5507, 0.2153, -0.0020, 0, 0, 0])
    movel(p[new_pose[0], new_pose[1], new_pose[2], current_pose[3], current_pose[4], current_pose[5]], a=0.8, v=0.2000)
    report_progress()
    set_digital_out(0, True)
    new_pose = pose_trans(tuft_coords, p[0.5507, 0.8347, -0.0020, 0, 0, 0])
    movel(p[new_pose[0], new_pose[1], new_pose[2], current_pose[3], current_pose[4], current_pose[5]], a=1.2, v=0.0600)
    report_progress()
    set_digital_out(0, False)
    new_pose = pose_trans(tuft_coords, p[0.5507, 0.8347, 0.1500, 0, 0, 0])
    movel(p[new_pose[0], new_pose[1], new_pose[2], current_pose[3], current_pose[4], current_pose[5]], a=0.8, v=0.2000)
    report_progress()
    new_pose = pose_trans(tuft_coords, p[0.5526, 0.2133, 0.1500, 0, 0, 0])
    movel(p[new_pose[0], new_pose[1], new_pose[2], current_pose[3], current_pose[4], current_pose[5]], a=1.2, v=0.2000)
    report_progress()
    new_pose = pose_trans(tuft_coords, p[0.5526, 0.2133, -0.0020, 0, 0, 0])
    movel(p[new_pose[0], new_pose[1], new_pose[2], current_pose[3], current_pose[4], current_pose[5]], a=0.8, v=0.2000)
    report_progress()
    set_digital_out(0, True)
    new_pose = pose_trans(tuft_coords, p[0.5526, 0.8367, -0.0020, 0, 0, 0])
    movel(p[new_pose[0], new_pose[1], new_pose[2], current_pose[3], current_pose[4], current_pose[5]], a=1.2, v=0.0600)
    report_progress()
    set_digital_out(0, False)
    new_pose = pose_trans(tuft_coords, p[0.5526, 0.8367, 0.1500, 0, 0, 0])
    movel(p[new_pose[0], new_pose[1], new_pose[2], current_pose[3], current_pose[4], current_pose[5]], a=0.8, v=0.2000)
    report_progress()
    new_pose = pose_trans(tuft_coords, p[0.5546, 0.2113, 0.1500, 0, 0, 0])
    movel(p[new_pose[0], new_pose[1], new_pose[2], current_pose[3], current_pose[4], current_pose[5]], a=1.2, v=0.2000)
    report_progress()
    new_pose = pose_trans(tuft_coords, p[0.5546, 0.2113, -0.0020, 0, 0, 0])
    movel(p[new_pose[0], new_pose[1], new_pose[2], current_pose[3], current_pose[4], current_pose[5]], a=0.8, v=0.2000)
    report_progress()
    set_digital_out(0, True)
    new_pose = pose_trans(tuft_coords, p[0.5546, 0.8387, -0.0020, 0, 0, 0])
    movel(p[new_pose[0], new_pose[1], new_pose[2], current_pose[3], current_pose[4], current_pose[5]], a=1.2, v=0.0600)
    report_progress()
    set_digital_out(0, False)
    new_pose = pose_trans(tuft_coords, p[0.5546, 0.8387, 0.1500, 0, 0, 0])
    movel(p[new_pose[0], new_pose[1], new_pose[2], current_pose[3], current_pose[4], current_pose[5]], a=0.8, v=0.2000)
    report_progress()
    new_pose = pose_trans(tuft_coords, p[0.5565, 0.2113, 0.1500, 0, 0, 0])
    movel(p[new_pose[0], new_pose[1], new_pose[2], current_pose[3], current_pose[4], current_pose[5]], a=1.2, v=0.2000)
    report_progress()
    new_pose = pose_trans(tuft_coords, p[0.5565, 0.2113, -0.0020, 0, 0, 0])
    movel(p[new_pose[0], new_pose[1], new_pose[2], current_pose[3], current_pose[4], current_pose[5]], a=0.8, v=0.2000)
    report_progress()
    set_digital_out(0, True)
    new_pose = pose_trans(tuft_coords, p[0.5565, 0.8387, -0.0020, 0, 0, 0])
    movel(p[new_pose[0], new_pose[1], new_pose[2], current_pose[3], current_pose[4], current_pose[5]], a=1.2, v=0.0600)
    report_progress()
    set_digital_out(0, False)
    new_pose = pose_trans(tuft_coords, p[0.5565, 0.8387, 0.1500, 0, 0, 0])
    movel(p[new_pose[0], new_pose[1], new_pose[2], current_pose[3], current_pose[4], current_pose[5]], a=0.8, v=0.2000)
    report_progress()
    new_pose = pose_trans(tuft_coords, p[0.5585, 0.2093, 0.1500, 0, 0, 0])
    movel(p[new_pose[0], new_pose[1], new_pose[2], current_pose[3], current_pose[4], current_pose[5]], a=1.2, v=0.2000)
    report_progress()
    new_pose = pose_trans(tuft_coords, p[0.5585, 0.2093, -0.0020, 0, 0, 0])
    movel(p[new_pose[0], new_pose[1], new_pose[2], current_pose[3], current_pose[4], current_pose[5]], a=0.8, v=0.2000)
    report_progress()
    set_digital_out(0, True)
    new_pose = pose_trans(tuft_coords, p[0.5585, 0.8407, -0.0020, 0, 0, 0])
    movel(p[new_pose[0], new_pose[1], new_pose[2], current_pose[3], current_pose[4], current_pose[5]], a=1.2, v=0.0600)
    report_progress()
    set_digital_out(0, False)
    new_pose = pose_trans(tuft_coords, p[0.5585, 0.8407, 0.1500, 0, 0, 0])
    movel(p[new_pose[0], new_pose[1], new_pose[2], current_pose[3], current_pose[4], current_pose[5]], a=0.8, v=0.2000)
    report_progress()
    new_pose = pose_trans(tuft_coords, p[0.5604, 0.2093, 0.1500, 0, 0, 0])
    movel(p[new_pose[0], new_pose[1], new_pose[2], current_pose[3], current_pose[4], current_pose[5]], a=1.2, v=0.2000)
    report_progress()
    new_pose = pose_trans(tuft_coords, p[0.5604, 0.2093, -0.0020, 0, 0, 0])
    movel(p[new_pose[0], new_pose[1], new_pose[2], current_pose[3], current_pose[4], current_pose[5]], a=0.8, v=0.2000)
    report_progress()
    set_digital_out(0, True)
    new_pose = pose_trans(tuft_coords, p[0.5604, 0.8407, -0.0020, 0, 0, 0])
    movel(p[new_pose[0], new_pose[1], new_pose[2], current_pose[3], current_pose[4], current_pose[5]], a=1.2, v=0.0600)
    report_progress()
    set_digital_out(0, False)
    new_pose = pose_trans(tuft_coords, p[0.5604, 0.8407, 0.1500, 0, 0, 0])
    movel(p[new_pose[0], new_pose[1], new_pose[2], current_pose[3], current_pose[4], current_pose[5]], a=0.8, v=0.2000)
    report_progress()
    new_pose = pose_trans(tuft_coords, p[0.5624, 0.2073, 0.1500, 0, 0, 0])
    movel(p[new_pose[0], new_pose[1], new_pose[2], current_pose[3], current_pose[4], current_pose[5]], a=1.2, v=0.2000)
    report_progress()
    new_pose = pose_trans(tuft_coords, p[0.5624, 0.2073, -0.0020, 0, 0, 0])
    movel(p[new_pose[0], new_pose[1], new_pose[2], current_pose[3], current_pose[4], current_pose[5]], a=0.8, v=0.2000)
    report_progress()
    set_digital_out(0, True)
    new_pose = pose_trans(tuft_coords, p[0.5624, 0.8427, -0.0020, 0, 0, 0])
    movel(p[new_pose[0], new_pose[1], new_pose[2], current_pose[3], current_pose[4], current_pose[5]], a=1.2, v=0.0600)
    report_progress()
    set_digital_out(0, False)
    new_pose = pose_trans(tuft_coords, p[0.5624, 0.8427, 0.1500, 0, 0, 0])
    movel(p[new_pose[0], new_pose[1], new_pose[2], current_pose[3], current_pose[4], current_pose[5]], a=0.8, v=0.2000)
    report_progress()
    new_pose = pose_trans(tuft_coords, p[0.5643, 0.2054, 0.1500, 0, 0, 0])
    movel(p[new_pose[0], new_pose[1], new_pose[2], current_pose[3], current_pose[4], current_pose[5]], a=1.2, v=0.2000)
    report_progress()
    new_pose = pose_trans(tuft_coords, p[0.5643, 0.2054, -0.0020, 0, 0, 0])
    movel(p[new_pose[0], new_pose[1], new_pose[2], current_pose[3], current_pose[4], current_pose[5]], a=0.8, v=0.2000)
    report_progress()
    set_digital_out(0, True)
    new_pose = pose_trans(tuft_coords, p[0.5643, 0.8446, -0.0020, 0, 0, 0])
    movel(p[new_pose[0], new_pose[1], new_pose[2], current_pose[3], current_pose[4], current_pose[5]], a=1.2, v=0.0600)
    report_progress()
    set_digital_out(0, False)
    new_pose = pose_trans(tuft_coords, p[0.5643, 0.8446, 0.1500, 0, 0, 0])
    movel(p[new_pose[0], new_pose[1], new_pose[2], current_pose[3], current_pose[4], current_pose[5]], a=0.8, v=0.2000)
    report_progress()
    new_pose = pose_trans(tuft_coords, p[0.5663, 0.2054, 0.1500, 0, 0, 0])
    movel(p[new_pose[0], new_pose[1], new_pose[2], current_pose[3], current_pose[4], current_pose[5]], a=1.2, v=0.2000)
    report_progress()
    new_pose = pose_trans(tuft_coords, p[0.5663, 0.2054, -0.0020, 0, 0, 0])
    movel(p[new_pose[0], new_pose[1], new_pose[2], current_pose[3], current_pose[4], current_pose[5]], a=0.8, v=0.2000)
    report_progress()
    set_digital_out(0, True)
    new_pose = pose_trans(tuft_coords, p[0.5663, 0.8446, -0.0020, 0, 0, 0])
    movel(p[new_pose[0], new_pose[1], new_pose[2], current_pose[3], current_pose[4], current_pose[5]], a=1.2, v=0.0600)
    report_progress()
    set_digital_out(0, False)
    new_pose = pose_trans(tuft_coords, p[0.5663, 0.8446, 0.1500, 0, 0, 0])
    movel(p[new_pose[0], new_pose[1], new_pose[2], current_pose[3], current_pose[4], current_pose[5]], a=0.8, v=0.2000)
    report_progress()
    new_pose = pose_trans(tuft_coords, p[0.5682, 0.2034, 0.1500, 0, 0, 0])
    movel(p[new_pose[0], new_pose[1], new_pose[2], current_pose[3], current_pose[4], current_pose[5]], a=1.2, v=0.2000)
    report_progress()
    new_pose = pose_trans(tuft_coords, p[0.5682, 0.2034, -0.0020, 0, 0, 0])
    movel(p[new_pose[0], new_pose[1], new_pose[2], current_pose[3], current_pose[4], current_pose[5]], a=0.8, v=0.2000)
    report_progress()
    set_digital_out(0, True)
    new_pose = pose_trans(tuft_coords, p[0.5682, 0.8466, -0.0020, 0, 0, 0])
    movel(p[new_pose[0], new_pose[1], new_pose[2], current_pose[3], current_pose[4], current_pose[5]], a=1.2, v=0.0600)
    report_progress()
    set_digital_out(0, False)
    new_pose = pose_trans(tuft_coords, p[0.5682, 0.8466, 0.1500, 0, 0, 0])
    movel(p[new_pose[0], new_pose[1], new_pose[2], current_pose[3], current_pose[4], current_pose[5]], a=0.8, v=0.2000)
    report_progress()
    new_pose = pose_trans(tuft_coords, p[0.5701, 0.2034, 0.1500, 0, 0, 0])
    movel(p[new_pose[0], new_pose[1], new_pose[2], current_pose[3], current_pose[4], current_pose[5]], a=1.2, v=0.2000)
    report_progress()
    new_pose = pose_trans(tuft_coords, p[0.5701, 0.2034, -0.0020, 0, 0, 0])
    movel(p[new_pose[0], new_pose[1], new_pose[2], current_pose[3], current_pose[4], current_pose[5]], a=0.8, v=0.2000)
    report_progress()
    set_digital_out(0, True)
    new_pose = pose_trans(tuft_coords, p[0.5701, 0.8466, -0.0020, 0, 0, 0])
    movel(p[new_pose[0], new_pose[1], new_pose[2], current_pose[3], current_pose[4], current_pose[5]], a=1.2, v=0.0600)
    report_progress()
    set_digital_out(0, False)
    new_pose = pose_trans(tuft_coords, p[0.5701, 0.8466, 0.1500, 0, 0, 0])
    movel(p[new_pose[0], new_pose[1], new_pose[2], current_pose[3], current_pose[4], current_pose[5]], a=0.8, v=0.2000)
    report_progress()
    new_pose = pose_trans(tuft_coords, p[0.5721, 0.2014, 0.1500, 0, 0, 0])
    movel(p[new_pose[0], new_pose[1], new_pose[2], current_pose[3], current_pose[4], current_pose[5]], a=1.2, v=0.2000)
    report_progress()
    new_pose = pose_trans(tuft_coords, p[0.5721, 0.2014, -0.0020, 0, 0, 0])
    movel(p[new_pose[0], new_pose[1], new_pose[2], current_pose[3], current_pose[4], current_pose[5]], a=0.8, v=0.2000)
    report_progress()
    set_digital_out(0, True)
    new_pose = pose_trans(tuft_coords, p[0.5721, 0.8486, -0.0020, 0, 0, 0])
    movel(p[new_pose[0], new_pose[1], new_pose[2], current_pose[3], current_pose[4], current_pose[5]], a=1.2, v=0.0600)
    report_progress()
    set_digital_out(0, False)
    new_pose = pose_trans(tuft_coords, p[0.5721, 0.8486, 0.1500, 0, 0, 0])
    movel(p[new_pose[0], new_pose[1], new_pose[2], current_pose[3], current_pose[4], current_pose[5]], a=0.8, v=0.2000)
    report_progress()
    new_pose = pose_trans(tuft_coords, p[0.5740, 0.1994, 0.1500, 0, 0, 0])
    movel(p[new_pose[0], new_pose[1], new_pose[2], current_pose[3], current_pose[4], current_pose[5]], a=1.2, v=0.2000)
    report_progress()
    new_pose = pose_trans(tuft_coords, p[0.5740, 0.1994, -0.0020, 0, 0, 0])
    movel(p[new_pose[0], new_pose[1], new_pose[2], current_pose[3], current_pose[4], current_pose[5]], a=0.8, v=0.2000)
    report_progress()
    set_digital_out(0, True)
    new_pose = pose_trans(tuft_coords, p[0.5740, 0.8506, -0.0020, 0, 0, 0])
    movel(p[new_pose[0], new_pose[1], new_pose[2], current_pose[3], current_pose[4], current_pose[5]], a=1.2, v=0.0600)
    report_progress()
    set_digital_out(0, False)
    new_pose = pose_trans(tuft_coords, p[0.5740, 0.8506, 0.1500, 0, 0, 0])
    movel(p[new_pose[0], new_pose[1], new_pose[2], current_pose[3], current_pose[4], current_pose[5]], a=0.8, v=0.2000)
    report_progress()
    new_pose = pose_trans(tuft_coords, p[0.5760, 0.1994, 0.1500, 0, 0, 0])
    movel(p[new_pose[0], new_pose[1], new_pose[2], current_pose[3], current_pose[4], current_pose[5]], a=1.2, v=0.2000)
    report_progress()
    new_pose = pose_trans(tuft_coords, p[0.5760, 0.1994, -0.0020, 0, 0, 0])
    movel(p[new_pose[0], new_pose[1], new_pose[2], current_pose[3], current_pose[4], current_pose[5]], a=0.8, v=0.2000)
    report_progress()
    set_digital_out(0, True)
    new_pose = pose_trans(tuft_coords, p[0.5760, 0.8506, -0.0020, 0, 0, 0])
    movel(p[new_pose[0], new_pose[1], new_pose[2], current_pose[3], current_pose[4], current_pose[5]], a=1.2, v=0.0600)
    report_progress()
    set_digital_out(0, False)
    new_pose = pose_trans(tuft_coords, p[0.5760, 0.8506, 0.1500, 0, 0, 0])
    movel(p[new_pose[0], new_pose[1], new_pose[2], current_pose[3], current_pose[4], current_pose[5]], a=0.8, v=0.2000)
    report_progress()
    new_pose = pose_trans(tuft_coords, p[0.5779, 0.1974, 0.1500, 0, 0, 0])
    movel(p[new_pose[0], new_pose[1], new_pose[2], current_pose[3], current_pose[4], current_pose[5]], a=1.2, v=0.2000)
    report_progress()
    new_pose = pose_trans(tuft_coords, p[0.5779, 0.1974, -0.0020, 0, 0, 0])
    movel(p[new_pose[0], new_pose[1], new_pose[2], current_pose[3], current_pose[4], current_pose[5]], a=0.8, v=0.2000)
    report_progress()
    set_digital_out(0, True)
    new_pose = pose_trans(tuft_coords, p[0.5779, 0.8526, -0.0020, 0, 0, 0])
    movel(p[new_pose[0], new_pose[1], new_pose[2], current_pose[3], current_pose[4], current_pose[5]], a=1.2, v=0.0600)
    report_progress()
    set_digital_out(0, False)
    new_pose = pose_trans(tuft_coords, p[0.5779, 0.8526, 0.1500, 0, 0, 0])
    movel(p[new_pose[0], new_pose[1], new_pose[2], current_pose[3], current_pose[4], current_pose[5]], a=0.8, v=0.2000)
    report_progress()
    new_pose = pose_trans(tuft_coords, p[0.5799, 0.1974, 0.1500, 0, 0, 0])
    movel(p[new_pose[0], new_pose[1], new_pose[2], current_pose[3], current_pose[4], current_pose[5]], a=1.2, v=0.2000)
    report_progress()
    new_pose = pose_trans(tuft_coords, p[0.5799, 0.1974, -0.0020, 0, 0, 0])
    movel(p[new_pose[0], new_pose[1], new_pose[2], current_pose[3], current_pose[4], current_pose[5]], a=0.8, v=0.2000)
    report_progress()
    set_digital_out(0, True)
    new_pose = pose_trans(tuft_coords, p[0.5799, 0.8526, -0.0020, 0, 0, 0])
    movel(p[new_pose[0], new_pose[1], new_pose[2], current_pose[3], current_pose[4], current_pose[5]], a=1.2, v=0.0600)
    report_progress()
    set_digital_out(0, False)
    new_pose = pose_trans(tuft_coords, p[0.5799, 0.8526, 0.1500, 0, 0, 0])
    movel(p[new_pose[0], new_pose[1], new_pose[2], current_pose[3], current_pose[4], current_pose[5]], a=0.8, v=0.2000)
    report_progress()
    new_pose = pose_trans(tuft_coords, p[0.5818, 0.1955, 0.1500, 0, 0, 0])
    movel(p[new_pose[0], new_pose[1], new_pose[2], current_pose[3], current_pose[4], current_pose[5]], a=1.2, v=0.2000)
    report_progress()
    new_pose = pose_trans(tuft_coords, p[0.5818, 0.1955, -0.0020, 0, 0, 0])
    movel(p[new_pose[0], new_pose[1], new_pose[2], current_pose[3], current_pose[4], current_pose[5]], a=0.8, v=0.2000)
    report_progress()
    set_digital_out(0, True)
    new_pose = pose_trans(tuft_coords, p[0.5818, 0.8545, -0.0020, 0, 0, 0])
    movel(p[new_pose[0], new_pose[1], new_pose[2], current_pose[3], current_pose[4], current_pose[5]], a=1.2, v=0.0600)
    report_progress()
    set_digital_out(0, False)
    new_pose = pose_trans(tuft_coords, p[0.5818, 0.8545, 0.1500, 0, 0, 0])
    movel(p[new_pose[0], new_pose[1], new_pose[2], current_pose[3], current_pose[4], current_pose[5]], a=0.8, v=0.2000)
    report_progress()
    new_pose = pose_trans(tuft_coords, p[0.5837, 0.1955, 0.1500, 0, 0, 0])
    movel(p[new_pose[0], new_pose[1], new_pose[2], current_pose[3], current_pose[4], current_pose[5]], a=1.2, v=0.2000)
    report_progress()
    new_pose = pose_trans(tuft_coords, p[0.5837, 0.1955, -0.0020, 0, 0, 0])
    movel(p[new_pose[0], new_pose[1], new_pose[2], current_pose[3], current_pose[4], current_pose[5]], a=0.8, v=0.2000)
    report_progress()
    set_digital_out(0, True)
    new_pose = pose_trans(tuft_coords, p[0.5837, 0.8545, -0.0020, 0, 0, 0])
    movel(p[new_pose[0], new_pose[1], new_pose[2], current_pose[3], current_pose[4], current_pose[5]], a=1.2, v=0.0600)
    report_progress()
    set_digital_out(0, False)
    new_pose = pose_trans(tuft_coords, p[0.5837, 0.8545, 0.1500, 0, 0, 0])
    movel(p[new_pose[0], new_pose[1], new_pose[2], current_pose[3], current_pose[4], current_pose[5]], a=0.8, v=0.2000)
    report_progress()
    new_pose = pose_trans(tuft_coords, p[0.5857, 0.1935, 0.1500, 0, 0, 0])
    movel(p[new_pose[0], new_pose[1], new_pose[2], current_pose[3], current_pose[4], current_pose[5]], a=1.2, v=0.2000)
    report_progress()
    new_pose = pose_trans(tuft_coords, p[0.5857, 0.1935, -0.0020, 0, 0, 0])
    movel(p[new_pose[0], new_pose[1], new_pose[2], current_pose[3], current_pose[4], current_pose[5]], a=0.8, v=0.2000)
    report_progress()
    set_digital_out(0, True)
    new_pose = pose_trans(tuft_coords, p[0.5857, 0.8565, -0.0020, 0, 0, 0])
    movel(p[new_pose[0], new_pose[1], new_pose[2], current_pose[3], current_pose[4], current_pose[5]], a=1.2, v=0.0600)
    report_progress()
    set_digital_out(0, False)
    new_pose = pose_trans(tuft_coords, p[0.5857, 0.8565, 0.1500, 0, 0, 0])
    movel(p[new_pose[0], new_pose[1], new_pose[2], current_pose[3], current_pose[4], current_pose[5]], a=0.8, v=0.2000)
    report_progress()
    new_pose = pose_trans(tuft_coords, p[0.5876, 0.1935, 0.1500, 0, 0, 0])
    movel(p[new_pose[0], new_pose[1], new_pose[2], current_pose[3], current_pose[4], current_pose[5]], a=1.2, v=0.2000)
    report_progress()
    new_pose = pose_trans(tuft_coords, p[0.5876, 0.1935, -0.0020, 0, 0, 0])
    movel(p[new_pose[0], new_pose[1], new_pose[2], current_pose[3], current_pose[4], current_pose[5]], a=0.8, v=0.2000)
    report_progress()
    set_digital_out(0, True)
    new_pose = pose_trans(tuft_coords, p[0.5876, 0.8565, -0.0020, 0, 0, 0])
    movel(p[new_pose[0], new_pose[1], new_pose[2], current_pose[3], current_pose[4], current_pose[5]], a=1.2, v=0.0600)
    report_progress()
    set_digital_out(0, False)
    new_pose = pose_trans(tuft_coords, p[0.5876, 0.8565, 0.1500, 0, 0, 0])
    movel(p[new_pose[0], new_pose[1], new_pose[2], current_pose[3], current_pose[4], current_pose[5]], a=0.8, v=0.2000)
    report_progress()
    new_pose = pose_trans(tuft_coords, p[0.5896, 0.1915, 0.1500, 0, 0, 0])
    movel(p[new_pose[0], new_pose[1], new_pose[2], current_pose[3], current_pose[4], current_pose[5]], a=1.2, v=0.2000)
    report_progress()
    new_pose = pose_trans(tuft_coords, p[0.5896, 0.1915, -0.0020, 0, 0, 0])
    movel(p[new_pose[0], new_pose[1], new_pose[2], current_pose[3], current_pose[4], current_pose[5]], a=0.8, v=0.2000)
    report_progress()
    set_digital_out(0, True)
    new_pose = pose_trans(tuft_coords, p[0.5896, 0.8585, -0.0020, 0, 0, 0])
    movel(p[new_pose[0], new_pose[1], new_pose[2], current_pose[3], current_pose[4], current_pose[5]], a=1.2, v=0.0600)
    report_progress()
    set_digital_out(0, False)
    new_pose = pose_trans(tuft_coords, p[0.5896, 0.8585, 0.1500, 0, 0, 0])
    movel(p[new_pose[0], new_pose[1], new_pose[2], current_pose[3], current_pose[4], current_pose[5]], a=0.8, v=0.2000)
    report_progress()
    new_pose = pose_trans(tuft_coords, p[0.5915, 0.1915, 0.1500, 0, 0, 0])
    movel(p[new_pose[0], new_pose[1], new_pose[2], current_pose[3], current_pose[4], current_pose[5]], a=1.2, v=0.2000)
    report_progress()
    new_pose = pose_trans(tuft_coords, p[0.5915, 0.1915, -0.0020, 0, 0, 0])
    movel(p[new_pose[0], new_pose[1], new_pose[2], current_pose[3], current_pose[4], current_pose[5]], a=0.8, v=0.2000)
